   // UNICODE_TO_GBK[42326] := 16#9DDE;
   // UNICODE_TO_GBK[42327] := 16#FA7B;
   // UNICODE_TO_GBK[42328] := 16#9DDF;
   // UNICODE_TO_GBK[42329] := 16#FA7C;
   // UNICODE_TO_GBK[42330] := 16#9DE0;
   // UNICODE_TO_GBK[42331] := 16#FA7D;
   // UNICODE_TO_GBK[42332] := 16#9DE1;
   // UNICODE_TO_GBK[42333] := 16#FA7E;
   // UNICODE_TO_GBK[42334] := 16#9DE2;
   // UNICODE_TO_GBK[42335] := 16#FA80;
   // UNICODE_TO_GBK[42336] := 16#9DE3;
   // UNICODE_TO_GBK[42337] := 16#FA81;
   // UNICODE_TO_GBK[42338] := 16#9DE4;
   // UNICODE_TO_GBK[42339] := 16#FA82;
   // UNICODE_TO_GBK[42340] := 16#9DE5;
   // UNICODE_TO_GBK[42341] := 16#FA83;
   // UNICODE_TO_GBK[42342] := 16#9DE6;
   // UNICODE_TO_GBK[42343] := 16#FA84;
   // UNICODE_TO_GBK[42344] := 16#9DE7;
   // UNICODE_TO_GBK[42345] := 16#FA85;
   // UNICODE_TO_GBK[42346] := 16#9DE8;
   // UNICODE_TO_GBK[42347] := 16#FA86;
   // UNICODE_TO_GBK[42348] := 16#9DE9;
   // UNICODE_TO_GBK[42349] := 16#FA87;
   // UNICODE_TO_GBK[42350] := 16#9DEA;
   // UNICODE_TO_GBK[42351] := 16#FA88;
   // UNICODE_TO_GBK[42352] := 16#9DEB;
   // UNICODE_TO_GBK[42353] := 16#FA89;
   // UNICODE_TO_GBK[42354] := 16#9DEC;
   // UNICODE_TO_GBK[42355] := 16#FA8A;
   // UNICODE_TO_GBK[42356] := 16#9DED;
   // UNICODE_TO_GBK[42357] := 16#FA8B;
   // UNICODE_TO_GBK[42358] := 16#9DEE;
   // UNICODE_TO_GBK[42359] := 16#FA8C;
   // UNICODE_TO_GBK[42360] := 16#9DEF;
   // UNICODE_TO_GBK[42361] := 16#FA8D;
   // UNICODE_TO_GBK[42362] := 16#9DF0;
   // UNICODE_TO_GBK[42363] := 16#FA8E;
   // UNICODE_TO_GBK[42364] := 16#9DF1;
   // UNICODE_TO_GBK[42365] := 16#FA8F;
   // UNICODE_TO_GBK[42366] := 16#9DF2;
   // UNICODE_TO_GBK[42367] := 16#FA90;
   // UNICODE_TO_GBK[42368] := 16#9DF3;
   // UNICODE_TO_GBK[42369] := 16#FA91;
   // UNICODE_TO_GBK[42370] := 16#9DF4;
   // UNICODE_TO_GBK[42371] := 16#FA92;
   // UNICODE_TO_GBK[42372] := 16#9DF5;
   // UNICODE_TO_GBK[42373] := 16#FA93;
   // UNICODE_TO_GBK[42374] := 16#9DF6;
   // UNICODE_TO_GBK[42375] := 16#FA94;
   // UNICODE_TO_GBK[42376] := 16#9DF7;
   // UNICODE_TO_GBK[42377] := 16#FA95;
   // UNICODE_TO_GBK[42378] := 16#9DF8;
   // UNICODE_TO_GBK[42379] := 16#FA96;
   // UNICODE_TO_GBK[42380] := 16#9DF9;
   // UNICODE_TO_GBK[42381] := 16#FA97;
   // UNICODE_TO_GBK[42382] := 16#9DFA;
   // UNICODE_TO_GBK[42383] := 16#FA98;
   // UNICODE_TO_GBK[42384] := 16#9DFB;
   // UNICODE_TO_GBK[42385] := 16#FA99;
   // UNICODE_TO_GBK[42386] := 16#9DFC;
   // UNICODE_TO_GBK[42387] := 16#FA9A;
   // UNICODE_TO_GBK[42388] := 16#9DFD;
   // UNICODE_TO_GBK[42389] := 16#FA9B;
   // UNICODE_TO_GBK[42390] := 16#9DFE;
   // UNICODE_TO_GBK[42391] := 16#FA9C;
   // UNICODE_TO_GBK[42392] := 16#9DFF;
   // UNICODE_TO_GBK[42393] := 16#FA9D;
   // UNICODE_TO_GBK[42394] := 16#9E00;
   // UNICODE_TO_GBK[42395] := 16#FA9E;
   // UNICODE_TO_GBK[42396] := 16#9E01;
   // UNICODE_TO_GBK[42397] := 16#FA9F;
   // UNICODE_TO_GBK[42398] := 16#9E02;
   // UNICODE_TO_GBK[42399] := 16#FAA0;
   // UNICODE_TO_GBK[42400] := 16#9E03;
   // UNICODE_TO_GBK[42401] := 16#FB40;
   // UNICODE_TO_GBK[42402] := 16#9E04;
   // UNICODE_TO_GBK[42403] := 16#FB41;
   // UNICODE_TO_GBK[42404] := 16#9E05;
   // UNICODE_TO_GBK[42405] := 16#FB42;
   // UNICODE_TO_GBK[42406] := 16#9E06;
   // UNICODE_TO_GBK[42407] := 16#FB43;
   // UNICODE_TO_GBK[42408] := 16#9E07;
   // UNICODE_TO_GBK[42409] := 16#FB44;
   // UNICODE_TO_GBK[42410] := 16#9E08;
   // UNICODE_TO_GBK[42411] := 16#FB45;
   // UNICODE_TO_GBK[42412] := 16#9E09;
   // UNICODE_TO_GBK[42413] := 16#FB46;
   // UNICODE_TO_GBK[42414] := 16#9E0A;
   // UNICODE_TO_GBK[42415] := 16#FB47;
   // UNICODE_TO_GBK[42416] := 16#9E0B;
   // UNICODE_TO_GBK[42417] := 16#FB48;
   // UNICODE_TO_GBK[42418] := 16#9E0C;
   // UNICODE_TO_GBK[42419] := 16#FB49;
   // UNICODE_TO_GBK[42420] := 16#9E0D;
   // UNICODE_TO_GBK[42421] := 16#FB4A;
   // UNICODE_TO_GBK[42422] := 16#9E0E;
   // UNICODE_TO_GBK[42423] := 16#FB4B;
   // UNICODE_TO_GBK[42424] := 16#9E0F;
   // UNICODE_TO_GBK[42425] := 16#FB4C;
   // UNICODE_TO_GBK[42426] := 16#9E10;
   // UNICODE_TO_GBK[42427] := 16#FB4D;
   // UNICODE_TO_GBK[42428] := 16#9E11;
   // UNICODE_TO_GBK[42429] := 16#FB4E;
   // UNICODE_TO_GBK[42430] := 16#9E12;
   // UNICODE_TO_GBK[42431] := 16#FB4F;
   // UNICODE_TO_GBK[42432] := 16#9E13;
   // UNICODE_TO_GBK[42433] := 16#FB50;
   // UNICODE_TO_GBK[42434] := 16#9E14;
   // UNICODE_TO_GBK[42435] := 16#FB51;
   // UNICODE_TO_GBK[42436] := 16#9E15;
   // UNICODE_TO_GBK[42437] := 16#FB52;
   // UNICODE_TO_GBK[42438] := 16#9E16;
   // UNICODE_TO_GBK[42439] := 16#FB53;
   // UNICODE_TO_GBK[42440] := 16#9E17;
   // UNICODE_TO_GBK[42441] := 16#FB54;
   // UNICODE_TO_GBK[42442] := 16#9E18;
   // UNICODE_TO_GBK[42443] := 16#FB55;
   // UNICODE_TO_GBK[42444] := 16#9E19;
   // UNICODE_TO_GBK[42445] := 16#FB56;
   // UNICODE_TO_GBK[42446] := 16#9E1A;
   // UNICODE_TO_GBK[42447] := 16#FB57;
   // UNICODE_TO_GBK[42448] := 16#9E1B;
   // UNICODE_TO_GBK[42449] := 16#FB58;
   // UNICODE_TO_GBK[42450] := 16#9E1C;
   // UNICODE_TO_GBK[42451] := 16#FB59;
   // UNICODE_TO_GBK[42452] := 16#9E1D;
   // UNICODE_TO_GBK[42453] := 16#FB5A;
   // UNICODE_TO_GBK[42454] := 16#9E1E;
   // UNICODE_TO_GBK[42455] := 16#FB5B;
   // UNICODE_TO_GBK[42456] := 16#9E1F;
   // UNICODE_TO_GBK[42457] := 16#C4F1;
   // UNICODE_TO_GBK[42458] := 16#9E20;
   // UNICODE_TO_GBK[42459] := 16#F0AF;
   // UNICODE_TO_GBK[42460] := 16#9E21;
   // UNICODE_TO_GBK[42461] := 16#BCA6;
   // UNICODE_TO_GBK[42462] := 16#9E22;
   // UNICODE_TO_GBK[42463] := 16#F0B0;
   // UNICODE_TO_GBK[42464] := 16#9E23;
   // UNICODE_TO_GBK[42465] := 16#C3F9;
   // UNICODE_TO_GBK[42466] := 16#9E24;
   // UNICODE_TO_GBK[42467] := 16#FB5C;
   // UNICODE_TO_GBK[42468] := 16#9E25;
   // UNICODE_TO_GBK[42469] := 16#C5B8;
   // UNICODE_TO_GBK[42470] := 16#9E26;
   // UNICODE_TO_GBK[42471] := 16#D1BB;
   // UNICODE_TO_GBK[42472] := 16#9E27;
   // UNICODE_TO_GBK[42473] := 16#FB5D;
   // UNICODE_TO_GBK[42474] := 16#9E28;
   // UNICODE_TO_GBK[42475] := 16#F0B1;
   // UNICODE_TO_GBK[42476] := 16#9E29;
   // UNICODE_TO_GBK[42477] := 16#F0B2;
   // UNICODE_TO_GBK[42478] := 16#9E2A;
   // UNICODE_TO_GBK[42479] := 16#F0B3;
   // UNICODE_TO_GBK[42480] := 16#9E2B;
   // UNICODE_TO_GBK[42481] := 16#F0B4;
   // UNICODE_TO_GBK[42482] := 16#9E2C;
   // UNICODE_TO_GBK[42483] := 16#F0B5;
   // UNICODE_TO_GBK[42484] := 16#9E2D;
   // UNICODE_TO_GBK[42485] := 16#D1BC;
   // UNICODE_TO_GBK[42486] := 16#9E2E;
   // UNICODE_TO_GBK[42487] := 16#FB5E;
   // UNICODE_TO_GBK[42488] := 16#9E2F;
   // UNICODE_TO_GBK[42489] := 16#D1EC;
   // UNICODE_TO_GBK[42490] := 16#9E30;
   // UNICODE_TO_GBK[42491] := 16#FB5F;
   // UNICODE_TO_GBK[42492] := 16#9E31;
   // UNICODE_TO_GBK[42493] := 16#F0B7;
   // UNICODE_TO_GBK[42494] := 16#9E32;
   // UNICODE_TO_GBK[42495] := 16#F0B6;
   // UNICODE_TO_GBK[42496] := 16#9E33;
   // UNICODE_TO_GBK[42497] := 16#D4A7;
   // UNICODE_TO_GBK[42498] := 16#9E34;
   // UNICODE_TO_GBK[42499] := 16#FB60;
   // UNICODE_TO_GBK[42500] := 16#9E35;
   // UNICODE_TO_GBK[42501] := 16#CDD2;
   // UNICODE_TO_GBK[42502] := 16#9E36;
   // UNICODE_TO_GBK[42503] := 16#F0B8;
   // UNICODE_TO_GBK[42504] := 16#9E37;
   // UNICODE_TO_GBK[42505] := 16#F0BA;
   // UNICODE_TO_GBK[42506] := 16#9E38;
   // UNICODE_TO_GBK[42507] := 16#F0B9;
   // UNICODE_TO_GBK[42508] := 16#9E39;
   // UNICODE_TO_GBK[42509] := 16#F0BB;
   // UNICODE_TO_GBK[42510] := 16#9E3A;
   // UNICODE_TO_GBK[42511] := 16#F0BC;
   // UNICODE_TO_GBK[42512] := 16#9E3B;
   // UNICODE_TO_GBK[42513] := 16#FB61;
   // UNICODE_TO_GBK[42514] := 16#9E3C;
   // UNICODE_TO_GBK[42515] := 16#FB62;
   // UNICODE_TO_GBK[42516] := 16#9E3D;
   // UNICODE_TO_GBK[42517] := 16#B8EB;
   // UNICODE_TO_GBK[42518] := 16#9E3E;
   // UNICODE_TO_GBK[42519] := 16#F0BD;
   // UNICODE_TO_GBK[42520] := 16#9E3F;
   // UNICODE_TO_GBK[42521] := 16#BAE8;
   // UNICODE_TO_GBK[42522] := 16#9E40;
   // UNICODE_TO_GBK[42523] := 16#FB63;
   // UNICODE_TO_GBK[42524] := 16#9E41;
   // UNICODE_TO_GBK[42525] := 16#F0BE;
   // UNICODE_TO_GBK[42526] := 16#9E42;
   // UNICODE_TO_GBK[42527] := 16#F0BF;
   // UNICODE_TO_GBK[42528] := 16#9E43;
   // UNICODE_TO_GBK[42529] := 16#BEE9;
   // UNICODE_TO_GBK[42530] := 16#9E44;
   // UNICODE_TO_GBK[42531] := 16#F0C0;
   // UNICODE_TO_GBK[42532] := 16#9E45;
   // UNICODE_TO_GBK[42533] := 16#B6EC;
   // UNICODE_TO_GBK[42534] := 16#9E46;
   // UNICODE_TO_GBK[42535] := 16#F0C1;
   // UNICODE_TO_GBK[42536] := 16#9E47;
   // UNICODE_TO_GBK[42537] := 16#F0C2;
   // UNICODE_TO_GBK[42538] := 16#9E48;
   // UNICODE_TO_GBK[42539] := 16#F0C3;
   // UNICODE_TO_GBK[42540] := 16#9E49;
   // UNICODE_TO_GBK[42541] := 16#F0C4;
   // UNICODE_TO_GBK[42542] := 16#9E4A;
   // UNICODE_TO_GBK[42543] := 16#C8B5;
   // UNICODE_TO_GBK[42544] := 16#9E4B;
   // UNICODE_TO_GBK[42545] := 16#F0C5;
   // UNICODE_TO_GBK[42546] := 16#9E4C;
   // UNICODE_TO_GBK[42547] := 16#F0C6;
   // UNICODE_TO_GBK[42548] := 16#9E4D;
   // UNICODE_TO_GBK[42549] := 16#FB64;
   // UNICODE_TO_GBK[42550] := 16#9E4E;
   // UNICODE_TO_GBK[42551] := 16#F0C7;
   // UNICODE_TO_GBK[42552] := 16#9E4F;
   // UNICODE_TO_GBK[42553] := 16#C5F4;
   // UNICODE_TO_GBK[42554] := 16#9E50;
   // UNICODE_TO_GBK[42555] := 16#FB65;
   // UNICODE_TO_GBK[42556] := 16#9E51;
   // UNICODE_TO_GBK[42557] := 16#F0C8;
   // UNICODE_TO_GBK[42558] := 16#9E52;
   // UNICODE_TO_GBK[42559] := 16#FB66;
   // UNICODE_TO_GBK[42560] := 16#9E53;
   // UNICODE_TO_GBK[42561] := 16#FB67;
   // UNICODE_TO_GBK[42562] := 16#9E54;
   // UNICODE_TO_GBK[42563] := 16#FB68;
   // UNICODE_TO_GBK[42564] := 16#9E55;
   // UNICODE_TO_GBK[42565] := 16#F0C9;
   // UNICODE_TO_GBK[42566] := 16#9E56;
   // UNICODE_TO_GBK[42567] := 16#FB69;
   // UNICODE_TO_GBK[42568] := 16#9E57;
   // UNICODE_TO_GBK[42569] := 16#F0CA;
   // UNICODE_TO_GBK[42570] := 16#9E58;
   // UNICODE_TO_GBK[42571] := 16#F7BD;
   // UNICODE_TO_GBK[42572] := 16#9E59;
   // UNICODE_TO_GBK[42573] := 16#FB6A;
   // UNICODE_TO_GBK[42574] := 16#9E5A;
   // UNICODE_TO_GBK[42575] := 16#F0CB;
   // UNICODE_TO_GBK[42576] := 16#9E5B;
   // UNICODE_TO_GBK[42577] := 16#F0CC;
   // UNICODE_TO_GBK[42578] := 16#9E5C;
   // UNICODE_TO_GBK[42579] := 16#F0CD;
   // UNICODE_TO_GBK[42580] := 16#9E5D;
   // UNICODE_TO_GBK[42581] := 16#FB6B;
   // UNICODE_TO_GBK[42582] := 16#9E5E;
   // UNICODE_TO_GBK[42583] := 16#F0CE;
   // UNICODE_TO_GBK[42584] := 16#9E5F;
   // UNICODE_TO_GBK[42585] := 16#FB6C;
   // UNICODE_TO_GBK[42586] := 16#9E60;
   // UNICODE_TO_GBK[42587] := 16#FB6D;
   // UNICODE_TO_GBK[42588] := 16#9E61;
   // UNICODE_TO_GBK[42589] := 16#FB6E;
   // UNICODE_TO_GBK[42590] := 16#9E62;
   // UNICODE_TO_GBK[42591] := 16#FB6F;
   // UNICODE_TO_GBK[42592] := 16#9E63;
   // UNICODE_TO_GBK[42593] := 16#F0CF;
   // UNICODE_TO_GBK[42594] := 16#9E64;
   // UNICODE_TO_GBK[42595] := 16#BAD7;
   // UNICODE_TO_GBK[42596] := 16#9E65;
   // UNICODE_TO_GBK[42597] := 16#FB70;
   // UNICODE_TO_GBK[42598] := 16#9E66;
   // UNICODE_TO_GBK[42599] := 16#F0D0;
   // UNICODE_TO_GBK[42600] := 16#9E67;
   // UNICODE_TO_GBK[42601] := 16#F0D1;
   // UNICODE_TO_GBK[42602] := 16#9E68;
   // UNICODE_TO_GBK[42603] := 16#F0D2;
   // UNICODE_TO_GBK[42604] := 16#9E69;
   // UNICODE_TO_GBK[42605] := 16#F0D3;
   // UNICODE_TO_GBK[42606] := 16#9E6A;
   // UNICODE_TO_GBK[42607] := 16#F0D4;
   // UNICODE_TO_GBK[42608] := 16#9E6B;
   // UNICODE_TO_GBK[42609] := 16#F0D5;
   // UNICODE_TO_GBK[42610] := 16#9E6C;
   // UNICODE_TO_GBK[42611] := 16#F0D6;
   // UNICODE_TO_GBK[42612] := 16#9E6D;
   // UNICODE_TO_GBK[42613] := 16#F0D8;
   // UNICODE_TO_GBK[42614] := 16#9E6E;
   // UNICODE_TO_GBK[42615] := 16#FB71;
   // UNICODE_TO_GBK[42616] := 16#9E6F;
   // UNICODE_TO_GBK[42617] := 16#FB72;
   // UNICODE_TO_GBK[42618] := 16#9E70;
   // UNICODE_TO_GBK[42619] := 16#D3A5;
   // UNICODE_TO_GBK[42620] := 16#9E71;
   // UNICODE_TO_GBK[42621] := 16#F0D7;
   // UNICODE_TO_GBK[42622] := 16#9E72;
   // UNICODE_TO_GBK[42623] := 16#FB73;
   // UNICODE_TO_GBK[42624] := 16#9E73;
   // UNICODE_TO_GBK[42625] := 16#F0D9;
   // UNICODE_TO_GBK[42626] := 16#9E74;
   // UNICODE_TO_GBK[42627] := 16#FB74;
   // UNICODE_TO_GBK[42628] := 16#9E75;
   // UNICODE_TO_GBK[42629] := 16#FB75;
   // UNICODE_TO_GBK[42630] := 16#9E76;
   // UNICODE_TO_GBK[42631] := 16#FB76;
   // UNICODE_TO_GBK[42632] := 16#9E77;
   // UNICODE_TO_GBK[42633] := 16#FB77;
   // UNICODE_TO_GBK[42634] := 16#9E78;
   // UNICODE_TO_GBK[42635] := 16#FB78;
   // UNICODE_TO_GBK[42636] := 16#9E79;
   // UNICODE_TO_GBK[42637] := 16#FB79;
   // UNICODE_TO_GBK[42638] := 16#9E7A;
   // UNICODE_TO_GBK[42639] := 16#FB7A;
   // UNICODE_TO_GBK[42640] := 16#9E7B;
   // UNICODE_TO_GBK[42641] := 16#FB7B;
   // UNICODE_TO_GBK[42642] := 16#9E7C;
   // UNICODE_TO_GBK[42643] := 16#FB7C;
   // UNICODE_TO_GBK[42644] := 16#9E7D;
   // UNICODE_TO_GBK[42645] := 16#FB7D;
   // UNICODE_TO_GBK[42646] := 16#9E7E;
   // UNICODE_TO_GBK[42647] := 16#F5BA;
   // UNICODE_TO_GBK[42648] := 16#9E7F;
   // UNICODE_TO_GBK[42649] := 16#C2B9;
   // UNICODE_TO_GBK[42650] := 16#9E80;
   // UNICODE_TO_GBK[42651] := 16#FB7E;
   // UNICODE_TO_GBK[42652] := 16#9E81;
   // UNICODE_TO_GBK[42653] := 16#FB80;
   // UNICODE_TO_GBK[42654] := 16#9E82;
   // UNICODE_TO_GBK[42655] := 16#F7E4;
   // UNICODE_TO_GBK[42656] := 16#9E83;
   // UNICODE_TO_GBK[42657] := 16#FB81;
   // UNICODE_TO_GBK[42658] := 16#9E84;
   // UNICODE_TO_GBK[42659] := 16#FB82;
   // UNICODE_TO_GBK[42660] := 16#9E85;
   // UNICODE_TO_GBK[42661] := 16#FB83;
   // UNICODE_TO_GBK[42662] := 16#9E86;
   // UNICODE_TO_GBK[42663] := 16#FB84;
   // UNICODE_TO_GBK[42664] := 16#9E87;
   // UNICODE_TO_GBK[42665] := 16#F7E5;
   // UNICODE_TO_GBK[42666] := 16#9E88;
   // UNICODE_TO_GBK[42667] := 16#F7E6;
   // UNICODE_TO_GBK[42668] := 16#9E89;
   // UNICODE_TO_GBK[42669] := 16#FB85;
   // UNICODE_TO_GBK[42670] := 16#9E8A;
   // UNICODE_TO_GBK[42671] := 16#FB86;
   // UNICODE_TO_GBK[42672] := 16#9E8B;
   // UNICODE_TO_GBK[42673] := 16#F7E7;
   // UNICODE_TO_GBK[42674] := 16#9E8C;
   // UNICODE_TO_GBK[42675] := 16#FB87;
   // UNICODE_TO_GBK[42676] := 16#9E8D;
   // UNICODE_TO_GBK[42677] := 16#FB88;
   // UNICODE_TO_GBK[42678] := 16#9E8E;
   // UNICODE_TO_GBK[42679] := 16#FB89;
   // UNICODE_TO_GBK[42680] := 16#9E8F;
   // UNICODE_TO_GBK[42681] := 16#FB8A;
   // UNICODE_TO_GBK[42682] := 16#9E90;
   // UNICODE_TO_GBK[42683] := 16#FB8B;
   // UNICODE_TO_GBK[42684] := 16#9E91;
   // UNICODE_TO_GBK[42685] := 16#FB8C;
   // UNICODE_TO_GBK[42686] := 16#9E92;
   // UNICODE_TO_GBK[42687] := 16#F7E8;
   // UNICODE_TO_GBK[42688] := 16#9E93;
   // UNICODE_TO_GBK[42689] := 16#C2B4;
   // UNICODE_TO_GBK[42690] := 16#9E94;
   // UNICODE_TO_GBK[42691] := 16#FB8D;
   // UNICODE_TO_GBK[42692] := 16#9E95;
   // UNICODE_TO_GBK[42693] := 16#FB8E;
   // UNICODE_TO_GBK[42694] := 16#9E96;
   // UNICODE_TO_GBK[42695] := 16#FB8F;
   // UNICODE_TO_GBK[42696] := 16#9E97;
   // UNICODE_TO_GBK[42697] := 16#FB90;
   // UNICODE_TO_GBK[42698] := 16#9E98;
   // UNICODE_TO_GBK[42699] := 16#FB91;
   // UNICODE_TO_GBK[42700] := 16#9E99;
   // UNICODE_TO_GBK[42701] := 16#FB92;
   // UNICODE_TO_GBK[42702] := 16#9E9A;
   // UNICODE_TO_GBK[42703] := 16#FB93;
   // UNICODE_TO_GBK[42704] := 16#9E9B;
   // UNICODE_TO_GBK[42705] := 16#FB94;
   // UNICODE_TO_GBK[42706] := 16#9E9C;
   // UNICODE_TO_GBK[42707] := 16#FB95;
   // UNICODE_TO_GBK[42708] := 16#9E9D;
   // UNICODE_TO_GBK[42709] := 16#F7EA;
   // UNICODE_TO_GBK[42710] := 16#9E9E;
   // UNICODE_TO_GBK[42711] := 16#FB96;
   // UNICODE_TO_GBK[42712] := 16#9E9F;
   // UNICODE_TO_GBK[42713] := 16#F7EB;
   // UNICODE_TO_GBK[42714] := 16#9EA0;
   // UNICODE_TO_GBK[42715] := 16#FB97;
   // UNICODE_TO_GBK[42716] := 16#9EA1;
   // UNICODE_TO_GBK[42717] := 16#FB98;
   // UNICODE_TO_GBK[42718] := 16#9EA2;
   // UNICODE_TO_GBK[42719] := 16#FB99;
   // UNICODE_TO_GBK[42720] := 16#9EA3;
   // UNICODE_TO_GBK[42721] := 16#FB9A;
   // UNICODE_TO_GBK[42722] := 16#9EA4;
   // UNICODE_TO_GBK[42723] := 16#FB9B;
   // UNICODE_TO_GBK[42724] := 16#9EA5;
   // UNICODE_TO_GBK[42725] := 16#FB9C;
   // UNICODE_TO_GBK[42726] := 16#9EA6;
   // UNICODE_TO_GBK[42727] := 16#C2F3;
   // UNICODE_TO_GBK[42728] := 16#9EA7;
   // UNICODE_TO_GBK[42729] := 16#FB9D;
   // UNICODE_TO_GBK[42730] := 16#9EA8;
   // UNICODE_TO_GBK[42731] := 16#FB9E;
   // UNICODE_TO_GBK[42732] := 16#9EA9;
   // UNICODE_TO_GBK[42733] := 16#FB9F;
   // UNICODE_TO_GBK[42734] := 16#9EAA;
   // UNICODE_TO_GBK[42735] := 16#FBA0;
   // UNICODE_TO_GBK[42736] := 16#9EAB;
   // UNICODE_TO_GBK[42737] := 16#FC40;
   // UNICODE_TO_GBK[42738] := 16#9EAC;
   // UNICODE_TO_GBK[42739] := 16#FC41;
   // UNICODE_TO_GBK[42740] := 16#9EAD;
   // UNICODE_TO_GBK[42741] := 16#FC42;
   // UNICODE_TO_GBK[42742] := 16#9EAE;
   // UNICODE_TO_GBK[42743] := 16#FC43;
   // UNICODE_TO_GBK[42744] := 16#9EAF;
   // UNICODE_TO_GBK[42745] := 16#FC44;
   // UNICODE_TO_GBK[42746] := 16#9EB0;
   // UNICODE_TO_GBK[42747] := 16#FC45;
   // UNICODE_TO_GBK[42748] := 16#9EB1;
   // UNICODE_TO_GBK[42749] := 16#FC46;
   // UNICODE_TO_GBK[42750] := 16#9EB2;
   // UNICODE_TO_GBK[42751] := 16#FC47;
   // UNICODE_TO_GBK[42752] := 16#9EB3;
   // UNICODE_TO_GBK[42753] := 16#FC48;
   // UNICODE_TO_GBK[42754] := 16#9EB4;
   // UNICODE_TO_GBK[42755] := 16#F4F0;
   // UNICODE_TO_GBK[42756] := 16#9EB5;
   // UNICODE_TO_GBK[42757] := 16#FC49;
   // UNICODE_TO_GBK[42758] := 16#9EB6;
   // UNICODE_TO_GBK[42759] := 16#FC4A;
   // UNICODE_TO_GBK[42760] := 16#9EB7;
   // UNICODE_TO_GBK[42761] := 16#FC4B;
   // UNICODE_TO_GBK[42762] := 16#9EB8;
   // UNICODE_TO_GBK[42763] := 16#F4EF;
   // UNICODE_TO_GBK[42764] := 16#9EB9;
   // UNICODE_TO_GBK[42765] := 16#FC4C;
   // UNICODE_TO_GBK[42766] := 16#9EBA;
   // UNICODE_TO_GBK[42767] := 16#FC4D;
   // UNICODE_TO_GBK[42768] := 16#9EBB;
   // UNICODE_TO_GBK[42769] := 16#C2E9;
   // UNICODE_TO_GBK[42770] := 16#9EBC;
   // UNICODE_TO_GBK[42771] := 16#FC4E;
   // UNICODE_TO_GBK[42772] := 16#9EBD;
   // UNICODE_TO_GBK[42773] := 16#F7E1;
   // UNICODE_TO_GBK[42774] := 16#9EBE;
   // UNICODE_TO_GBK[42775] := 16#F7E2;
   // UNICODE_TO_GBK[42776] := 16#9EBF;
   // UNICODE_TO_GBK[42777] := 16#FC4F;
   // UNICODE_TO_GBK[42778] := 16#9EC0;
   // UNICODE_TO_GBK[42779] := 16#FC50;
   // UNICODE_TO_GBK[42780] := 16#9EC1;
   // UNICODE_TO_GBK[42781] := 16#FC51;
   // UNICODE_TO_GBK[42782] := 16#9EC2;
   // UNICODE_TO_GBK[42783] := 16#FC52;
   // UNICODE_TO_GBK[42784] := 16#9EC3;
   // UNICODE_TO_GBK[42785] := 16#FC53;
   // UNICODE_TO_GBK[42786] := 16#9EC4;
   // UNICODE_TO_GBK[42787] := 16#BBC6;
   // UNICODE_TO_GBK[42788] := 16#9EC5;
   // UNICODE_TO_GBK[42789] := 16#FC54;
   // UNICODE_TO_GBK[42790] := 16#9EC6;
   // UNICODE_TO_GBK[42791] := 16#FC55;
   // UNICODE_TO_GBK[42792] := 16#9EC7;
   // UNICODE_TO_GBK[42793] := 16#FC56;
   // UNICODE_TO_GBK[42794] := 16#9EC8;
   // UNICODE_TO_GBK[42795] := 16#FC57;
   // UNICODE_TO_GBK[42796] := 16#9EC9;
   // UNICODE_TO_GBK[42797] := 16#D9E4;
   // UNICODE_TO_GBK[42798] := 16#9ECA;
   // UNICODE_TO_GBK[42799] := 16#FC58;
   // UNICODE_TO_GBK[42800] := 16#9ECB;
   // UNICODE_TO_GBK[42801] := 16#FC59;
   // UNICODE_TO_GBK[42802] := 16#9ECC;
   // UNICODE_TO_GBK[42803] := 16#FC5A;
   // UNICODE_TO_GBK[42804] := 16#9ECD;
   // UNICODE_TO_GBK[42805] := 16#CAF2;
   // UNICODE_TO_GBK[42806] := 16#9ECE;
   // UNICODE_TO_GBK[42807] := 16#C0E8;
   // UNICODE_TO_GBK[42808] := 16#9ECF;
   // UNICODE_TO_GBK[42809] := 16#F0A4;
   // UNICODE_TO_GBK[42810] := 16#9ED0;
   // UNICODE_TO_GBK[42811] := 16#FC5B;
   // UNICODE_TO_GBK[42812] := 16#9ED1;
   // UNICODE_TO_GBK[42813] := 16#BADA;
   // UNICODE_TO_GBK[42814] := 16#9ED2;
   // UNICODE_TO_GBK[42815] := 16#FC5C;
   // UNICODE_TO_GBK[42816] := 16#9ED3;
   // UNICODE_TO_GBK[42817] := 16#FC5D;
   // UNICODE_TO_GBK[42818] := 16#9ED4;
   // UNICODE_TO_GBK[42819] := 16#C7AD;
   // UNICODE_TO_GBK[42820] := 16#9ED5;
   // UNICODE_TO_GBK[42821] := 16#FC5E;
   // UNICODE_TO_GBK[42822] := 16#9ED6;
   // UNICODE_TO_GBK[42823] := 16#FC5F;
   // UNICODE_TO_GBK[42824] := 16#9ED7;
   // UNICODE_TO_GBK[42825] := 16#FC60;
   // UNICODE_TO_GBK[42826] := 16#9ED8;
   // UNICODE_TO_GBK[42827] := 16#C4AC;
   // UNICODE_TO_GBK[42828] := 16#9ED9;
   // UNICODE_TO_GBK[42829] := 16#FC61;
   // UNICODE_TO_GBK[42830] := 16#9EDA;
   // UNICODE_TO_GBK[42831] := 16#FC62;
   // UNICODE_TO_GBK[42832] := 16#9EDB;
   // UNICODE_TO_GBK[42833] := 16#F7EC;
   // UNICODE_TO_GBK[42834] := 16#9EDC;
   // UNICODE_TO_GBK[42835] := 16#F7ED;
   // UNICODE_TO_GBK[42836] := 16#9EDD;
   // UNICODE_TO_GBK[42837] := 16#F7EE;
   // UNICODE_TO_GBK[42838] := 16#9EDE;
   // UNICODE_TO_GBK[42839] := 16#FC63;
   // UNICODE_TO_GBK[42840] := 16#9EDF;
   // UNICODE_TO_GBK[42841] := 16#F7F0;
   // UNICODE_TO_GBK[42842] := 16#9EE0;
   // UNICODE_TO_GBK[42843] := 16#F7EF;
   // UNICODE_TO_GBK[42844] := 16#9EE1;
   // UNICODE_TO_GBK[42845] := 16#FC64;
   // UNICODE_TO_GBK[42846] := 16#9EE2;
   // UNICODE_TO_GBK[42847] := 16#F7F1;
   // UNICODE_TO_GBK[42848] := 16#9EE3;
   // UNICODE_TO_GBK[42849] := 16#FC65;
   // UNICODE_TO_GBK[42850] := 16#9EE4;
   // UNICODE_TO_GBK[42851] := 16#FC66;
   // UNICODE_TO_GBK[42852] := 16#9EE5;
   // UNICODE_TO_GBK[42853] := 16#F7F4;
   // UNICODE_TO_GBK[42854] := 16#9EE6;
   // UNICODE_TO_GBK[42855] := 16#FC67;
   // UNICODE_TO_GBK[42856] := 16#9EE7;
   // UNICODE_TO_GBK[42857] := 16#F7F3;
   // UNICODE_TO_GBK[42858] := 16#9EE8;
   // UNICODE_TO_GBK[42859] := 16#FC68;
   // UNICODE_TO_GBK[42860] := 16#9EE9;
   // UNICODE_TO_GBK[42861] := 16#F7F2;
   // UNICODE_TO_GBK[42862] := 16#9EEA;
   // UNICODE_TO_GBK[42863] := 16#F7F5;
   // UNICODE_TO_GBK[42864] := 16#9EEB;
   // UNICODE_TO_GBK[42865] := 16#FC69;
   // UNICODE_TO_GBK[42866] := 16#9EEC;
   // UNICODE_TO_GBK[42867] := 16#FC6A;
   // UNICODE_TO_GBK[42868] := 16#9EED;
   // UNICODE_TO_GBK[42869] := 16#FC6B;
   // UNICODE_TO_GBK[42870] := 16#9EEE;
   // UNICODE_TO_GBK[42871] := 16#FC6C;
   // UNICODE_TO_GBK[42872] := 16#9EEF;
   // UNICODE_TO_GBK[42873] := 16#F7F6;
   // UNICODE_TO_GBK[42874] := 16#9EF0;
   // UNICODE_TO_GBK[42875] := 16#FC6D;
   // UNICODE_TO_GBK[42876] := 16#9EF1;
   // UNICODE_TO_GBK[42877] := 16#FC6E;
   // UNICODE_TO_GBK[42878] := 16#9EF2;
   // UNICODE_TO_GBK[42879] := 16#FC6F;
   // UNICODE_TO_GBK[42880] := 16#9EF3;
   // UNICODE_TO_GBK[42881] := 16#FC70;
   // UNICODE_TO_GBK[42882] := 16#9EF4;
   // UNICODE_TO_GBK[42883] := 16#FC71;
   // UNICODE_TO_GBK[42884] := 16#9EF5;
   // UNICODE_TO_GBK[42885] := 16#FC72;
   // UNICODE_TO_GBK[42886] := 16#9EF6;
   // UNICODE_TO_GBK[42887] := 16#FC73;
   // UNICODE_TO_GBK[42888] := 16#9EF7;
   // UNICODE_TO_GBK[42889] := 16#FC74;
   // UNICODE_TO_GBK[42890] := 16#9EF8;
   // UNICODE_TO_GBK[42891] := 16#FC75;
   // UNICODE_TO_GBK[42892] := 16#9EF9;
   // UNICODE_TO_GBK[42893] := 16#EDE9;
   // UNICODE_TO_GBK[42894] := 16#9EFA;
   // UNICODE_TO_GBK[42895] := 16#FC76;
   // UNICODE_TO_GBK[42896] := 16#9EFB;
   // UNICODE_TO_GBK[42897] := 16#EDEA;
   // UNICODE_TO_GBK[42898] := 16#9EFC;
   // UNICODE_TO_GBK[42899] := 16#EDEB;
   // UNICODE_TO_GBK[42900] := 16#9EFD;
   // UNICODE_TO_GBK[42901] := 16#FC77;
   // UNICODE_TO_GBK[42902] := 16#9EFE;
   // UNICODE_TO_GBK[42903] := 16#F6BC;
   // UNICODE_TO_GBK[42904] := 16#9EFF;
   // UNICODE_TO_GBK[42905] := 16#FC78;
   // UNICODE_TO_GBK[42906] := 16#9F00;
   // UNICODE_TO_GBK[42907] := 16#FC79;
   // UNICODE_TO_GBK[42908] := 16#9F01;
   // UNICODE_TO_GBK[42909] := 16#FC7A;
   // UNICODE_TO_GBK[42910] := 16#9F02;
   // UNICODE_TO_GBK[42911] := 16#FC7B;
   // UNICODE_TO_GBK[42912] := 16#9F03;
   // UNICODE_TO_GBK[42913] := 16#FC7C;
   // UNICODE_TO_GBK[42914] := 16#9F04;
   // UNICODE_TO_GBK[42915] := 16#FC7D;
   // UNICODE_TO_GBK[42916] := 16#9F05;
   // UNICODE_TO_GBK[42917] := 16#FC7E;
   // UNICODE_TO_GBK[42918] := 16#9F06;
   // UNICODE_TO_GBK[42919] := 16#FC80;
   // UNICODE_TO_GBK[42920] := 16#9F07;
   // UNICODE_TO_GBK[42921] := 16#FC81;
   // UNICODE_TO_GBK[42922] := 16#9F08;
   // UNICODE_TO_GBK[42923] := 16#FC82;
   // UNICODE_TO_GBK[42924] := 16#9F09;
   // UNICODE_TO_GBK[42925] := 16#FC83;
   // UNICODE_TO_GBK[42926] := 16#9F0A;
   // UNICODE_TO_GBK[42927] := 16#FC84;
   // UNICODE_TO_GBK[42928] := 16#9F0B;
   // UNICODE_TO_GBK[42929] := 16#F6BD;
   // UNICODE_TO_GBK[42930] := 16#9F0C;
   // UNICODE_TO_GBK[42931] := 16#FC85;
   // UNICODE_TO_GBK[42932] := 16#9F0D;
   // UNICODE_TO_GBK[42933] := 16#F6BE;
   // UNICODE_TO_GBK[42934] := 16#9F0E;
   // UNICODE_TO_GBK[42935] := 16#B6A6;
   // UNICODE_TO_GBK[42936] := 16#9F0F;
   // UNICODE_TO_GBK[42937] := 16#FC86;
   // UNICODE_TO_GBK[42938] := 16#9F10;
   // UNICODE_TO_GBK[42939] := 16#D8BE;
   // UNICODE_TO_GBK[42940] := 16#9F11;
   // UNICODE_TO_GBK[42941] := 16#FC87;
   // UNICODE_TO_GBK[42942] := 16#9F12;
   // UNICODE_TO_GBK[42943] := 16#FC88;
   // UNICODE_TO_GBK[42944] := 16#9F13;
   // UNICODE_TO_GBK[42945] := 16#B9C4;
   // UNICODE_TO_GBK[42946] := 16#9F14;
   // UNICODE_TO_GBK[42947] := 16#FC89;
   // UNICODE_TO_GBK[42948] := 16#9F15;
   // UNICODE_TO_GBK[42949] := 16#FC8A;
   // UNICODE_TO_GBK[42950] := 16#9F16;
   // UNICODE_TO_GBK[42951] := 16#FC8B;
   // UNICODE_TO_GBK[42952] := 16#9F17;
   // UNICODE_TO_GBK[42953] := 16#D8BB;
   // UNICODE_TO_GBK[42954] := 16#9F18;
   // UNICODE_TO_GBK[42955] := 16#FC8C;
   // UNICODE_TO_GBK[42956] := 16#9F19;
   // UNICODE_TO_GBK[42957] := 16#DCB1;
   // UNICODE_TO_GBK[42958] := 16#9F1A;
   // UNICODE_TO_GBK[42959] := 16#FC8D;
   // UNICODE_TO_GBK[42960] := 16#9F1B;
   // UNICODE_TO_GBK[42961] := 16#FC8E;
   // UNICODE_TO_GBK[42962] := 16#9F1C;
   // UNICODE_TO_GBK[42963] := 16#FC8F;
   // UNICODE_TO_GBK[42964] := 16#9F1D;
   // UNICODE_TO_GBK[42965] := 16#FC90;
   // UNICODE_TO_GBK[42966] := 16#9F1E;
   // UNICODE_TO_GBK[42967] := 16#FC91;
   // UNICODE_TO_GBK[42968] := 16#9F1F;
   // UNICODE_TO_GBK[42969] := 16#FC92;
   // UNICODE_TO_GBK[42970] := 16#9F20;
   // UNICODE_TO_GBK[42971] := 16#CAF3;
   // UNICODE_TO_GBK[42972] := 16#9F21;
   // UNICODE_TO_GBK[42973] := 16#FC93;
   // UNICODE_TO_GBK[42974] := 16#9F22;
   // UNICODE_TO_GBK[42975] := 16#F7F7;
   // UNICODE_TO_GBK[42976] := 16#9F23;
   // UNICODE_TO_GBK[42977] := 16#FC94;
   // UNICODE_TO_GBK[42978] := 16#9F24;
   // UNICODE_TO_GBK[42979] := 16#FC95;
   // UNICODE_TO_GBK[42980] := 16#9F25;
   // UNICODE_TO_GBK[42981] := 16#FC96;
   // UNICODE_TO_GBK[42982] := 16#9F26;
   // UNICODE_TO_GBK[42983] := 16#FC97;
   // UNICODE_TO_GBK[42984] := 16#9F27;
   // UNICODE_TO_GBK[42985] := 16#FC98;
   // UNICODE_TO_GBK[42986] := 16#9F28;
   // UNICODE_TO_GBK[42987] := 16#FC99;
   // UNICODE_TO_GBK[42988] := 16#9F29;
   // UNICODE_TO_GBK[42989] := 16#FC9A;
   // UNICODE_TO_GBK[42990] := 16#9F2A;
   // UNICODE_TO_GBK[42991] := 16#FC9B;
   // UNICODE_TO_GBK[42992] := 16#9F2B;
   // UNICODE_TO_GBK[42993] := 16#FC9C;
   // UNICODE_TO_GBK[42994] := 16#9F2C;
   // UNICODE_TO_GBK[42995] := 16#F7F8;
   // UNICODE_TO_GBK[42996] := 16#9F2D;
   // UNICODE_TO_GBK[42997] := 16#FC9D;
   // UNICODE_TO_GBK[42998] := 16#9F2E;
   // UNICODE_TO_GBK[42999] := 16#FC9E;
   // UNICODE_TO_GBK[43000] := 16#9F2F;
   // UNICODE_TO_GBK[43001] := 16#F7F9;
   // UNICODE_TO_GBK[43002] := 16#9F30;
   // UNICODE_TO_GBK[43003] := 16#FC9F;
   // UNICODE_TO_GBK[43004] := 16#9F31;
   // UNICODE_TO_GBK[43005] := 16#FCA0;
   // UNICODE_TO_GBK[43006] := 16#9F32;
   // UNICODE_TO_GBK[43007] := 16#FD40;
   // UNICODE_TO_GBK[43008] := 16#9F33;
   // UNICODE_TO_GBK[43009] := 16#FD41;
   // UNICODE_TO_GBK[43010] := 16#9F34;
   // UNICODE_TO_GBK[43011] := 16#FD42;
   // UNICODE_TO_GBK[43012] := 16#9F35;
   // UNICODE_TO_GBK[43013] := 16#FD43;
   // UNICODE_TO_GBK[43014] := 16#9F36;
   // UNICODE_TO_GBK[43015] := 16#FD44;
   // UNICODE_TO_GBK[43016] := 16#9F37;
   // UNICODE_TO_GBK[43017] := 16#F7FB;
   // UNICODE_TO_GBK[43018] := 16#9F38;
   // UNICODE_TO_GBK[43019] := 16#FD45;
   // UNICODE_TO_GBK[43020] := 16#9F39;
   // UNICODE_TO_GBK[43021] := 16#F7FA;
   // UNICODE_TO_GBK[43022] := 16#9F3A;
   // UNICODE_TO_GBK[43023] := 16#FD46;
   // UNICODE_TO_GBK[43024] := 16#9F3B;
   // UNICODE_TO_GBK[43025] := 16#B1C7;
   // UNICODE_TO_GBK[43026] := 16#9F3C;
   // UNICODE_TO_GBK[43027] := 16#FD47;
   // UNICODE_TO_GBK[43028] := 16#9F3D;
   // UNICODE_TO_GBK[43029] := 16#F7FC;
   // UNICODE_TO_GBK[43030] := 16#9F3E;
   // UNICODE_TO_GBK[43031] := 16#F7FD;
   // UNICODE_TO_GBK[43032] := 16#9F3F;
   // UNICODE_TO_GBK[43033] := 16#FD48;
   // UNICODE_TO_GBK[43034] := 16#9F40;
   // UNICODE_TO_GBK[43035] := 16#FD49;
   // UNICODE_TO_GBK[43036] := 16#9F41;
   // UNICODE_TO_GBK[43037] := 16#FD4A;
   // UNICODE_TO_GBK[43038] := 16#9F42;
   // UNICODE_TO_GBK[43039] := 16#FD4B;
   // UNICODE_TO_GBK[43040] := 16#9F43;
   // UNICODE_TO_GBK[43041] := 16#FD4C;
   // UNICODE_TO_GBK[43042] := 16#9F44;
   // UNICODE_TO_GBK[43043] := 16#F7FE;
   // UNICODE_TO_GBK[43044] := 16#9F45;
   // UNICODE_TO_GBK[43045] := 16#FD4D;
   // UNICODE_TO_GBK[43046] := 16#9F46;
   // UNICODE_TO_GBK[43047] := 16#FD4E;
   // UNICODE_TO_GBK[43048] := 16#9F47;
   // UNICODE_TO_GBK[43049] := 16#FD4F;
   // UNICODE_TO_GBK[43050] := 16#9F48;
   // UNICODE_TO_GBK[43051] := 16#FD50;
   // UNICODE_TO_GBK[43052] := 16#9F49;
   // UNICODE_TO_GBK[43053] := 16#FD51;
   // UNICODE_TO_GBK[43054] := 16#9F4A;
   // UNICODE_TO_GBK[43055] := 16#FD52;
   // UNICODE_TO_GBK[43056] := 16#9F4B;
   // UNICODE_TO_GBK[43057] := 16#FD53;
   // UNICODE_TO_GBK[43058] := 16#9F4C;
   // UNICODE_TO_GBK[43059] := 16#FD54;
   // UNICODE_TO_GBK[43060] := 16#9F4D;
   // UNICODE_TO_GBK[43061] := 16#FD55;
   // UNICODE_TO_GBK[43062] := 16#9F4E;
   // UNICODE_TO_GBK[43063] := 16#FD56;
   // UNICODE_TO_GBK[43064] := 16#9F4F;
   // UNICODE_TO_GBK[43065] := 16#FD57;
   // UNICODE_TO_GBK[43066] := 16#9F50;
   // UNICODE_TO_GBK[43067] := 16#C6EB;
   // UNICODE_TO_GBK[43068] := 16#9F51;
   // UNICODE_TO_GBK[43069] := 16#ECB4;
   // UNICODE_TO_GBK[43070] := 16#9F52;
   // UNICODE_TO_GBK[43071] := 16#FD58;
   // UNICODE_TO_GBK[43072] := 16#9F53;
   // UNICODE_TO_GBK[43073] := 16#FD59;
   // UNICODE_TO_GBK[43074] := 16#9F54;
   // UNICODE_TO_GBK[43075] := 16#FD5A;
   // UNICODE_TO_GBK[43076] := 16#9F55;
   // UNICODE_TO_GBK[43077] := 16#FD5B;
   // UNICODE_TO_GBK[43078] := 16#9F56;
   // UNICODE_TO_GBK[43079] := 16#FD5C;
   // UNICODE_TO_GBK[43080] := 16#9F57;
   // UNICODE_TO_GBK[43081] := 16#FD5D;
   // UNICODE_TO_GBK[43082] := 16#9F58;
   // UNICODE_TO_GBK[43083] := 16#FD5E;
   // UNICODE_TO_GBK[43084] := 16#9F59;
   // UNICODE_TO_GBK[43085] := 16#FD5F;
   // UNICODE_TO_GBK[43086] := 16#9F5A;
   // UNICODE_TO_GBK[43087] := 16#FD60;
   // UNICODE_TO_GBK[43088] := 16#9F5B;
   // UNICODE_TO_GBK[43089] := 16#FD61;
   // UNICODE_TO_GBK[43090] := 16#9F5C;
   // UNICODE_TO_GBK[43091] := 16#FD62;
   // UNICODE_TO_GBK[43092] := 16#9F5D;
   // UNICODE_TO_GBK[43093] := 16#FD63;
   // UNICODE_TO_GBK[43094] := 16#9F5E;
   // UNICODE_TO_GBK[43095] := 16#FD64;
   // UNICODE_TO_GBK[43096] := 16#9F5F;
   // UNICODE_TO_GBK[43097] := 16#FD65;
   // UNICODE_TO_GBK[43098] := 16#9F60;
   // UNICODE_TO_GBK[43099] := 16#FD66;
   // UNICODE_TO_GBK[43100] := 16#9F61;
   // UNICODE_TO_GBK[43101] := 16#FD67;
   // UNICODE_TO_GBK[43102] := 16#9F62;
   // UNICODE_TO_GBK[43103] := 16#FD68;
   // UNICODE_TO_GBK[43104] := 16#9F63;
   // UNICODE_TO_GBK[43105] := 16#FD69;
   // UNICODE_TO_GBK[43106] := 16#9F64;
   // UNICODE_TO_GBK[43107] := 16#FD6A;
   // UNICODE_TO_GBK[43108] := 16#9F65;
   // UNICODE_TO_GBK[43109] := 16#FD6B;
   // UNICODE_TO_GBK[43110] := 16#9F66;
   // UNICODE_TO_GBK[43111] := 16#FD6C;
   // UNICODE_TO_GBK[43112] := 16#9F67;
   // UNICODE_TO_GBK[43113] := 16#FD6D;
   // UNICODE_TO_GBK[43114] := 16#9F68;
   // UNICODE_TO_GBK[43115] := 16#FD6E;
   // UNICODE_TO_GBK[43116] := 16#9F69;
   // UNICODE_TO_GBK[43117] := 16#FD6F;
   // UNICODE_TO_GBK[43118] := 16#9F6A;
   // UNICODE_TO_GBK[43119] := 16#FD70;
   // UNICODE_TO_GBK[43120] := 16#9F6B;
   // UNICODE_TO_GBK[43121] := 16#FD71;
   // UNICODE_TO_GBK[43122] := 16#9F6C;
   // UNICODE_TO_GBK[43123] := 16#FD72;
   // UNICODE_TO_GBK[43124] := 16#9F6D;
   // UNICODE_TO_GBK[43125] := 16#FD73;
   // UNICODE_TO_GBK[43126] := 16#9F6E;
   // UNICODE_TO_GBK[43127] := 16#FD74;
   // UNICODE_TO_GBK[43128] := 16#9F6F;
   // UNICODE_TO_GBK[43129] := 16#FD75;
   // UNICODE_TO_GBK[43130] := 16#9F70;
   // UNICODE_TO_GBK[43131] := 16#FD76;
   // UNICODE_TO_GBK[43132] := 16#9F71;
   // UNICODE_TO_GBK[43133] := 16#FD77;
   // UNICODE_TO_GBK[43134] := 16#9F72;
   // UNICODE_TO_GBK[43135] := 16#FD78;
   // UNICODE_TO_GBK[43136] := 16#9F73;
   // UNICODE_TO_GBK[43137] := 16#FD79;
   // UNICODE_TO_GBK[43138] := 16#9F74;
   // UNICODE_TO_GBK[43139] := 16#FD7A;
   // UNICODE_TO_GBK[43140] := 16#9F75;
   // UNICODE_TO_GBK[43141] := 16#FD7B;
   // UNICODE_TO_GBK[43142] := 16#9F76;
   // UNICODE_TO_GBK[43143] := 16#FD7C;
   // UNICODE_TO_GBK[43144] := 16#9F77;
   // UNICODE_TO_GBK[43145] := 16#FD7D;
   // UNICODE_TO_GBK[43146] := 16#9F78;
   // UNICODE_TO_GBK[43147] := 16#FD7E;
   // UNICODE_TO_GBK[43148] := 16#9F79;
   // UNICODE_TO_GBK[43149] := 16#FD80;
   // UNICODE_TO_GBK[43150] := 16#9F7A;
   // UNICODE_TO_GBK[43151] := 16#FD81;
   // UNICODE_TO_GBK[43152] := 16#9F7B;
   // UNICODE_TO_GBK[43153] := 16#FD82;
   // UNICODE_TO_GBK[43154] := 16#9F7C;
   // UNICODE_TO_GBK[43155] := 16#FD83;
   // UNICODE_TO_GBK[43156] := 16#9F7D;
   // UNICODE_TO_GBK[43157] := 16#FD84;
   // UNICODE_TO_GBK[43158] := 16#9F7E;
   // UNICODE_TO_GBK[43159] := 16#FD85;
   // UNICODE_TO_GBK[43160] := 16#9F7F;
   // UNICODE_TO_GBK[43161] := 16#B3DD;
   // UNICODE_TO_GBK[43162] := 16#9F80;
   // UNICODE_TO_GBK[43163] := 16#F6B3;
   // UNICODE_TO_GBK[43164] := 16#9F81;
   // UNICODE_TO_GBK[43165] := 16#FD86;
   // UNICODE_TO_GBK[43166] := 16#9F82;
   // UNICODE_TO_GBK[43167] := 16#FD87;
   // UNICODE_TO_GBK[43168] := 16#9F83;
   // UNICODE_TO_GBK[43169] := 16#F6B4;
   // UNICODE_TO_GBK[43170] := 16#9F84;
   // UNICODE_TO_GBK[43171] := 16#C1E4;
   // UNICODE_TO_GBK[43172] := 16#9F85;
   // UNICODE_TO_GBK[43173] := 16#F6B5;
   // UNICODE_TO_GBK[43174] := 16#9F86;
   // UNICODE_TO_GBK[43175] := 16#F6B6;
   // UNICODE_TO_GBK[43176] := 16#9F87;
   // UNICODE_TO_GBK[43177] := 16#F6B7;
   // UNICODE_TO_GBK[43178] := 16#9F88;
   // UNICODE_TO_GBK[43179] := 16#F6B8;
   // UNICODE_TO_GBK[43180] := 16#9F89;
   // UNICODE_TO_GBK[43181] := 16#F6B9;
   // UNICODE_TO_GBK[43182] := 16#9F8A;
   // UNICODE_TO_GBK[43183] := 16#F6BA;
   // UNICODE_TO_GBK[43184] := 16#9F8B;
   // UNICODE_TO_GBK[43185] := 16#C8A3;
   // UNICODE_TO_GBK[43186] := 16#9F8C;
   // UNICODE_TO_GBK[43187] := 16#F6BB;
   // UNICODE_TO_GBK[43188] := 16#9F8D;
   // UNICODE_TO_GBK[43189] := 16#FD88;
   // UNICODE_TO_GBK[43190] := 16#9F8E;
   // UNICODE_TO_GBK[43191] := 16#FD89;
   // UNICODE_TO_GBK[43192] := 16#9F8F;
   // UNICODE_TO_GBK[43193] := 16#FD8A;
   // UNICODE_TO_GBK[43194] := 16#9F90;
   // UNICODE_TO_GBK[43195] := 16#FD8B;
   // UNICODE_TO_GBK[43196] := 16#9F91;
   // UNICODE_TO_GBK[43197] := 16#FD8C;
   // UNICODE_TO_GBK[43198] := 16#9F92;
   // UNICODE_TO_GBK[43199] := 16#FD8D;
   // UNICODE_TO_GBK[43200] := 16#9F93;
   // UNICODE_TO_GBK[43201] := 16#FD8E;
   // UNICODE_TO_GBK[43202] := 16#9F94;
   // UNICODE_TO_GBK[43203] := 16#FD8F;
   // UNICODE_TO_GBK[43204] := 16#9F95;
   // UNICODE_TO_GBK[43205] := 16#FD90;
   // UNICODE_TO_GBK[43206] := 16#9F96;
   // UNICODE_TO_GBK[43207] := 16#FD91;
   // UNICODE_TO_GBK[43208] := 16#9F97;
   // UNICODE_TO_GBK[43209] := 16#FD92;
   // UNICODE_TO_GBK[43210] := 16#9F98;
   // UNICODE_TO_GBK[43211] := 16#FD93;
   // UNICODE_TO_GBK[43212] := 16#9F99;
   // UNICODE_TO_GBK[43213] := 16#C1FA;
   // UNICODE_TO_GBK[43214] := 16#9F9A;
   // UNICODE_TO_GBK[43215] := 16#B9A8;
   // UNICODE_TO_GBK[43216] := 16#9F9B;
   // UNICODE_TO_GBK[43217] := 16#EDE8;
   // UNICODE_TO_GBK[43218] := 16#9F9C;
   // UNICODE_TO_GBK[43219] := 16#FD94;
   // UNICODE_TO_GBK[43220] := 16#9F9D;
   // UNICODE_TO_GBK[43221] := 16#FD95;
   // UNICODE_TO_GBK[43222] := 16#9F9E;
   // UNICODE_TO_GBK[43223] := 16#FD96;
   // UNICODE_TO_GBK[43224] := 16#9F9F;
   // UNICODE_TO_GBK[43225] := 16#B9EA;
   // UNICODE_TO_GBK[43226] := 16#9FA0;
   // UNICODE_TO_GBK[43227] := 16#D9DF;
   // UNICODE_TO_GBK[43228] := 16#9FA1;
   // UNICODE_TO_GBK[43229] := 16#FD97;
   // UNICODE_TO_GBK[43230] := 16#9FA2;
   // UNICODE_TO_GBK[43231] := 16#FD98;
   // UNICODE_TO_GBK[43232] := 16#9FA3;
   // UNICODE_TO_GBK[43233] := 16#FD99;
   // UNICODE_TO_GBK[43234] := 16#9FA4;
   // UNICODE_TO_GBK[43235] := 16#FD9A;
   // UNICODE_TO_GBK[43236] := 16#9FA5;
   // UNICODE_TO_GBK[43237] := 16#FD9B;
   // UNICODE_TO_GBK[43238] := 16#F92C;
   // UNICODE_TO_GBK[43239] := 16#FD9C;
   // UNICODE_TO_GBK[43240] := 16#F979;
   // UNICODE_TO_GBK[43241] := 16#FD9D;
   // UNICODE_TO_GBK[43242] := 16#F995;
   // UNICODE_TO_GBK[43243] := 16#FD9E;
   // UNICODE_TO_GBK[43244] := 16#F9E7;
   // UNICODE_TO_GBK[43245] := 16#FD9F;
   // UNICODE_TO_GBK[43246] := 16#F9F1;
   // UNICODE_TO_GBK[43247] := 16#FDA0;
   // UNICODE_TO_GBK[43248] := 16#FA0C;
   // UNICODE_TO_GBK[43249] := 16#FE40;
   // UNICODE_TO_GBK[43250] := 16#FA0D;
   // UNICODE_TO_GBK[43251] := 16#FE41;
   // UNICODE_TO_GBK[43252] := 16#FA0E;
   // UNICODE_TO_GBK[43253] := 16#FE42;
   // UNICODE_TO_GBK[43254] := 16#FA0F;
   // UNICODE_TO_GBK[43255] := 16#FE43;
   // UNICODE_TO_GBK[43256] := 16#FA11;
   // UNICODE_TO_GBK[43257] := 16#FE44;
   // UNICODE_TO_GBK[43258] := 16#FA13;
   // UNICODE_TO_GBK[43259] := 16#FE45;
   // UNICODE_TO_GBK[43260] := 16#FA14;
   // UNICODE_TO_GBK[43261] := 16#FE46;
   // UNICODE_TO_GBK[43262] := 16#FA18;
   // UNICODE_TO_GBK[43263] := 16#FE47;
   // UNICODE_TO_GBK[43264] := 16#FA1F;
   // UNICODE_TO_GBK[43265] := 16#FE48;
   // UNICODE_TO_GBK[43266] := 16#FA20;
   // UNICODE_TO_GBK[43267] := 16#FE49;
   // UNICODE_TO_GBK[43268] := 16#FA21;
   // UNICODE_TO_GBK[43269] := 16#FE4A;
   // UNICODE_TO_GBK[43270] := 16#FA23;
   // UNICODE_TO_GBK[43271] := 16#FE4B;
   // UNICODE_TO_GBK[43272] := 16#FA24;
   // UNICODE_TO_GBK[43273] := 16#FE4C;
   // UNICODE_TO_GBK[43274] := 16#FA27;
   // UNICODE_TO_GBK[43275] := 16#FE4D;
   // UNICODE_TO_GBK[43276] := 16#FA28;
   // UNICODE_TO_GBK[43277] := 16#FE4E;
   // UNICODE_TO_GBK[43278] := 16#FA29;
   // UNICODE_TO_GBK[43279] := 16#FE4F;
   // UNICODE_TO_GBK[43280] := 16#FE30;
   // UNICODE_TO_GBK[43281] := 16#A955;
   // UNICODE_TO_GBK[43282] := 16#FE31;
   // UNICODE_TO_GBK[43283] := 16#A6F2;
   // UNICODE_TO_GBK[43284] := 16#FE33;
   // UNICODE_TO_GBK[43285] := 16#A6F4;
   // UNICODE_TO_GBK[43286] := 16#FE34;
   // UNICODE_TO_GBK[43287] := 16#A6F5;
   // UNICODE_TO_GBK[43288] := 16#FE35;
   // UNICODE_TO_GBK[43289] := 16#A6E0;
   // UNICODE_TO_GBK[43290] := 16#FE36;
   // UNICODE_TO_GBK[43291] := 16#A6E1;
   // UNICODE_TO_GBK[43292] := 16#FE37;
   // UNICODE_TO_GBK[43293] := 16#A6F0;
   // UNICODE_TO_GBK[43294] := 16#FE38;
   // UNICODE_TO_GBK[43295] := 16#A6F1;
   // UNICODE_TO_GBK[43296] := 16#FE39;
   // UNICODE_TO_GBK[43297] := 16#A6E2;
   // UNICODE_TO_GBK[43298] := 16#FE3A;
   // UNICODE_TO_GBK[43299] := 16#A6E3;
   // UNICODE_TO_GBK[43300] := 16#FE3B;
   // UNICODE_TO_GBK[43301] := 16#A6EE;
   // UNICODE_TO_GBK[43302] := 16#FE3C;
   // UNICODE_TO_GBK[43303] := 16#A6EF;
   // UNICODE_TO_GBK[43304] := 16#FE3D;
   // UNICODE_TO_GBK[43305] := 16#A6E6;
   // UNICODE_TO_GBK[43306] := 16#FE3E;
   // UNICODE_TO_GBK[43307] := 16#A6E7;
   // UNICODE_TO_GBK[43308] := 16#FE3F;
   // UNICODE_TO_GBK[43309] := 16#A6E4;
   // UNICODE_TO_GBK[43310] := 16#FE40;
   // UNICODE_TO_GBK[43311] := 16#A6E5;
   // UNICODE_TO_GBK[43312] := 16#FE41;
   // UNICODE_TO_GBK[43313] := 16#A6E8;
   // UNICODE_TO_GBK[43314] := 16#FE42;
   // UNICODE_TO_GBK[43315] := 16#A6E9;
   // UNICODE_TO_GBK[43316] := 16#FE43;
   // UNICODE_TO_GBK[43317] := 16#A6EA;
   // UNICODE_TO_GBK[43318] := 16#FE44;
   // UNICODE_TO_GBK[43319] := 16#A6EB;
   // UNICODE_TO_GBK[43320] := 16#FE49;
   // UNICODE_TO_GBK[43321] := 16#A968;
   // UNICODE_TO_GBK[43322] := 16#FE4A;
   // UNICODE_TO_GBK[43323] := 16#A969;
   // UNICODE_TO_GBK[43324] := 16#FE4B;
   // UNICODE_TO_GBK[43325] := 16#A96A;
   // UNICODE_TO_GBK[43326] := 16#FE4C;
   // UNICODE_TO_GBK[43327] := 16#A96B;
   // UNICODE_TO_GBK[43328] := 16#FE4D;
   // UNICODE_TO_GBK[43329] := 16#A96C;
   // UNICODE_TO_GBK[43330] := 16#FE4E;
   // UNICODE_TO_GBK[43331] := 16#A96D;
   // UNICODE_TO_GBK[43332] := 16#FE4F;
   // UNICODE_TO_GBK[43333] := 16#A96E;
   // UNICODE_TO_GBK[43334] := 16#FE50;
   // UNICODE_TO_GBK[43335] := 16#A96F;
   // UNICODE_TO_GBK[43336] := 16#FE51;
   // UNICODE_TO_GBK[43337] := 16#A970;
   // UNICODE_TO_GBK[43338] := 16#FE52;
   // UNICODE_TO_GBK[43339] := 16#A971;
   // UNICODE_TO_GBK[43340] := 16#FE54;
   // UNICODE_TO_GBK[43341] := 16#A972;
   // UNICODE_TO_GBK[43342] := 16#FE55;
   // UNICODE_TO_GBK[43343] := 16#A973;
   // UNICODE_TO_GBK[43344] := 16#FE56;
   // UNICODE_TO_GBK[43345] := 16#A974;
   // UNICODE_TO_GBK[43346] := 16#FE57;
   // UNICODE_TO_GBK[43347] := 16#A975;
   // UNICODE_TO_GBK[43348] := 16#FE59;
   // UNICODE_TO_GBK[43349] := 16#A976;
   // UNICODE_TO_GBK[43350] := 16#FE5A;
   // UNICODE_TO_GBK[43351] := 16#A977;
   // UNICODE_TO_GBK[43352] := 16#FE5B;
   // UNICODE_TO_GBK[43353] := 16#A978;
   // UNICODE_TO_GBK[43354] := 16#FE5C;
   // UNICODE_TO_GBK[43355] := 16#A979;
   // UNICODE_TO_GBK[43356] := 16#FE5D;
   // UNICODE_TO_GBK[43357] := 16#A97A;
   // UNICODE_TO_GBK[43358] := 16#FE5E;
   // UNICODE_TO_GBK[43359] := 16#A97B;
   // UNICODE_TO_GBK[43360] := 16#FE5F;
   // UNICODE_TO_GBK[43361] := 16#A97C;
   // UNICODE_TO_GBK[43362] := 16#FE60;
   // UNICODE_TO_GBK[43363] := 16#A97D;
   // UNICODE_TO_GBK[43364] := 16#FE61;
   // UNICODE_TO_GBK[43365] := 16#A97E;
   // UNICODE_TO_GBK[43366] := 16#FE62;
   // UNICODE_TO_GBK[43367] := 16#A980;
   // UNICODE_TO_GBK[43368] := 16#FE63;
   // UNICODE_TO_GBK[43369] := 16#A981;
   // UNICODE_TO_GBK[43370] := 16#FE64;
   // UNICODE_TO_GBK[43371] := 16#A982;
   // UNICODE_TO_GBK[43372] := 16#FE65;
   // UNICODE_TO_GBK[43373] := 16#A983;
   // UNICODE_TO_GBK[43374] := 16#FE66;
   // UNICODE_TO_GBK[43375] := 16#A984;
   // UNICODE_TO_GBK[43376] := 16#FE68;
   // UNICODE_TO_GBK[43377] := 16#A985;
   // UNICODE_TO_GBK[43378] := 16#FE69;
   // UNICODE_TO_GBK[43379] := 16#A986;
   // UNICODE_TO_GBK[43380] := 16#FE6A;
   // UNICODE_TO_GBK[43381] := 16#A987;
   // UNICODE_TO_GBK[43382] := 16#FE6B;
   // UNICODE_TO_GBK[43383] := 16#A988;
   // UNICODE_TO_GBK[43384] := 16#FF01;
   // UNICODE_TO_GBK[43385] := 16#A3A1;
   // UNICODE_TO_GBK[43386] := 16#FF02;
   // UNICODE_TO_GBK[43387] := 16#A3A2;
   // UNICODE_TO_GBK[43388] := 16#FF03;
   // UNICODE_TO_GBK[43389] := 16#A3A3;
   // UNICODE_TO_GBK[43390] := 16#FF04;
   // UNICODE_TO_GBK[43391] := 16#A1E7;
   // UNICODE_TO_GBK[43392] := 16#FF05;
   // UNICODE_TO_GBK[43393] := 16#A3A5;
   // UNICODE_TO_GBK[43394] := 16#FF06;
   // UNICODE_TO_GBK[43395] := 16#A3A6;
   // UNICODE_TO_GBK[43396] := 16#FF07;
   // UNICODE_TO_GBK[43397] := 16#A3A7;
   // UNICODE_TO_GBK[43398] := 16#FF08;
   // UNICODE_TO_GBK[43399] := 16#A3A8;
   // UNICODE_TO_GBK[43400] := 16#FF09;
   // UNICODE_TO_GBK[43401] := 16#A3A9;
   // UNICODE_TO_GBK[43402] := 16#FF0A;
   // UNICODE_TO_GBK[43403] := 16#A3AA;
   // UNICODE_TO_GBK[43404] := 16#FF0B;
   // UNICODE_TO_GBK[43405] := 16#A3AB;
   // UNICODE_TO_GBK[43406] := 16#FF0C;
   // UNICODE_TO_GBK[43407] := 16#A3AC;
   // UNICODE_TO_GBK[43408] := 16#FF0D;
   // UNICODE_TO_GBK[43409] := 16#A3AD;
   // UNICODE_TO_GBK[43410] := 16#FF0E;
   // UNICODE_TO_GBK[43411] := 16#A3AE;
   // UNICODE_TO_GBK[43412] := 16#FF0F;
   // UNICODE_TO_GBK[43413] := 16#A3AF;
   // UNICODE_TO_GBK[43414] := 16#FF10;
   // UNICODE_TO_GBK[43415] := 16#A3B0;
   // UNICODE_TO_GBK[43416] := 16#FF11;
   // UNICODE_TO_GBK[43417] := 16#A3B1;
   // UNICODE_TO_GBK[43418] := 16#FF12;
   // UNICODE_TO_GBK[43419] := 16#A3B2;
   // UNICODE_TO_GBK[43420] := 16#FF13;
   // UNICODE_TO_GBK[43421] := 16#A3B3;
   // UNICODE_TO_GBK[43422] := 16#FF14;
   // UNICODE_TO_GBK[43423] := 16#A3B4;
   // UNICODE_TO_GBK[43424] := 16#FF15;
   // UNICODE_TO_GBK[43425] := 16#A3B5;
   // UNICODE_TO_GBK[43426] := 16#FF16;
   // UNICODE_TO_GBK[43427] := 16#A3B6;
   // UNICODE_TO_GBK[43428] := 16#FF17;
   // UNICODE_TO_GBK[43429] := 16#A3B7;
   // UNICODE_TO_GBK[43430] := 16#FF18;
   // UNICODE_TO_GBK[43431] := 16#A3B8;
   // UNICODE_TO_GBK[43432] := 16#FF19;
   // UNICODE_TO_GBK[43433] := 16#A3B9;
   // UNICODE_TO_GBK[43434] := 16#FF1A;
   // UNICODE_TO_GBK[43435] := 16#A3BA;
   // UNICODE_TO_GBK[43436] := 16#FF1B;
   // UNICODE_TO_GBK[43437] := 16#A3BB;
   // UNICODE_TO_GBK[43438] := 16#FF1C;
   // UNICODE_TO_GBK[43439] := 16#A3BC;
   // UNICODE_TO_GBK[43440] := 16#FF1D;
   // UNICODE_TO_GBK[43441] := 16#A3BD;
   // UNICODE_TO_GBK[43442] := 16#FF1E;
   // UNICODE_TO_GBK[43443] := 16#A3BE;
   // UNICODE_TO_GBK[43444] := 16#FF1F;
   // UNICODE_TO_GBK[43445] := 16#A3BF;
   // UNICODE_TO_GBK[43446] := 16#FF20;
   // UNICODE_TO_GBK[43447] := 16#A3C0;
   // UNICODE_TO_GBK[43448] := 16#FF21;
   // UNICODE_TO_GBK[43449] := 16#A3C1;
   // UNICODE_TO_GBK[43450] := 16#FF22;
   // UNICODE_TO_GBK[43451] := 16#A3C2;
   // UNICODE_TO_GBK[43452] := 16#FF23;
   // UNICODE_TO_GBK[43453] := 16#A3C3;
   // UNICODE_TO_GBK[43454] := 16#FF24;
   // UNICODE_TO_GBK[43455] := 16#A3C4;
   // UNICODE_TO_GBK[43456] := 16#FF25;
   // UNICODE_TO_GBK[43457] := 16#A3C5;
   // UNICODE_TO_GBK[43458] := 16#FF26;
   // UNICODE_TO_GBK[43459] := 16#A3C6;
   // UNICODE_TO_GBK[43460] := 16#FF27;
   // UNICODE_TO_GBK[43461] := 16#A3C7;
   // UNICODE_TO_GBK[43462] := 16#FF28;
   // UNICODE_TO_GBK[43463] := 16#A3C8;
   // UNICODE_TO_GBK[43464] := 16#FF29;
   // UNICODE_TO_GBK[43465] := 16#A3C9;
   // UNICODE_TO_GBK[43466] := 16#FF2A;
   // UNICODE_TO_GBK[43467] := 16#A3CA;
   // UNICODE_TO_GBK[43468] := 16#FF2B;
   // UNICODE_TO_GBK[43469] := 16#A3CB;
   // UNICODE_TO_GBK[43470] := 16#FF2C;
   // UNICODE_TO_GBK[43471] := 16#A3CC;
   // UNICODE_TO_GBK[43472] := 16#FF2D;
   // UNICODE_TO_GBK[43473] := 16#A3CD;
   // UNICODE_TO_GBK[43474] := 16#FF2E;
   // UNICODE_TO_GBK[43475] := 16#A3CE;
   // UNICODE_TO_GBK[43476] := 16#FF2F;
   // UNICODE_TO_GBK[43477] := 16#A3CF;
   // UNICODE_TO_GBK[43478] := 16#FF30;
   // UNICODE_TO_GBK[43479] := 16#A3D0;
   // UNICODE_TO_GBK[43480] := 16#FF31;
   // UNICODE_TO_GBK[43481] := 16#A3D1;
   // UNICODE_TO_GBK[43482] := 16#FF32;
   // UNICODE_TO_GBK[43483] := 16#A3D2;
   // UNICODE_TO_GBK[43484] := 16#FF33;
   // UNICODE_TO_GBK[43485] := 16#A3D3;
   // UNICODE_TO_GBK[43486] := 16#FF34;
   // UNICODE_TO_GBK[43487] := 16#A3D4;
   // UNICODE_TO_GBK[43488] := 16#FF35;
   // UNICODE_TO_GBK[43489] := 16#A3D5;
   // UNICODE_TO_GBK[43490] := 16#FF36;
   // UNICODE_TO_GBK[43491] := 16#A3D6;
   // UNICODE_TO_GBK[43492] := 16#FF37;
   // UNICODE_TO_GBK[43493] := 16#A3D7;
   // UNICODE_TO_GBK[43494] := 16#FF38;
   // UNICODE_TO_GBK[43495] := 16#A3D8;
   // UNICODE_TO_GBK[43496] := 16#FF39;
   // UNICODE_TO_GBK[43497] := 16#A3D9;
   // UNICODE_TO_GBK[43498] := 16#FF3A;
   // UNICODE_TO_GBK[43499] := 16#A3DA;
   // UNICODE_TO_GBK[43500] := 16#FF3B;
   // UNICODE_TO_GBK[43501] := 16#A3DB;
   // UNICODE_TO_GBK[43502] := 16#FF3C;
   // UNICODE_TO_GBK[43503] := 16#A3DC;
   // UNICODE_TO_GBK[43504] := 16#FF3D;
   // UNICODE_TO_GBK[43505] := 16#A3DD;
   // UNICODE_TO_GBK[43506] := 16#FF3E;
   // UNICODE_TO_GBK[43507] := 16#A3DE;
   // UNICODE_TO_GBK[43508] := 16#FF3F;
   // UNICODE_TO_GBK[43509] := 16#A3DF;
   // UNICODE_TO_GBK[43510] := 16#FF40;
   // UNICODE_TO_GBK[43511] := 16#A3E0;
   // UNICODE_TO_GBK[43512] := 16#FF41;
   // UNICODE_TO_GBK[43513] := 16#A3E1;
   // UNICODE_TO_GBK[43514] := 16#FF42;
   // UNICODE_TO_GBK[43515] := 16#A3E2;
   // UNICODE_TO_GBK[43516] := 16#FF43;
   // UNICODE_TO_GBK[43517] := 16#A3E3;
   // UNICODE_TO_GBK[43518] := 16#FF44;
   // UNICODE_TO_GBK[43519] := 16#A3E4;
   // UNICODE_TO_GBK[43520] := 16#FF45;
   // UNICODE_TO_GBK[43521] := 16#A3E5;
   // UNICODE_TO_GBK[43522] := 16#FF46;
   // UNICODE_TO_GBK[43523] := 16#A3E6;
   // UNICODE_TO_GBK[43524] := 16#FF47;
   // UNICODE_TO_GBK[43525] := 16#A3E7;
   // UNICODE_TO_GBK[43526] := 16#FF48;
   // UNICODE_TO_GBK[43527] := 16#A3E8;
   // UNICODE_TO_GBK[43528] := 16#FF49;
   // UNICODE_TO_GBK[43529] := 16#A3E9;
   // UNICODE_TO_GBK[43530] := 16#FF4A;
   // UNICODE_TO_GBK[43531] := 16#A3EA;
   // UNICODE_TO_GBK[43532] := 16#FF4B;
   // UNICODE_TO_GBK[43533] := 16#A3EB;
   // UNICODE_TO_GBK[43534] := 16#FF4C;
   // UNICODE_TO_GBK[43535] := 16#A3EC;
   // UNICODE_TO_GBK[43536] := 16#FF4D;
   // UNICODE_TO_GBK[43537] := 16#A3ED;
   // UNICODE_TO_GBK[43538] := 16#FF4E;
   // UNICODE_TO_GBK[43539] := 16#A3EE;
   // UNICODE_TO_GBK[43540] := 16#FF4F;
   // UNICODE_TO_GBK[43541] := 16#A3EF;
   // UNICODE_TO_GBK[43542] := 16#FF50;
   // UNICODE_TO_GBK[43543] := 16#A3F0;
   // UNICODE_TO_GBK[43544] := 16#FF51;
   // UNICODE_TO_GBK[43545] := 16#A3F1;
   // UNICODE_TO_GBK[43546] := 16#FF52;
   // UNICODE_TO_GBK[43547] := 16#A3F2;
   // UNICODE_TO_GBK[43548] := 16#FF53;
   // UNICODE_TO_GBK[43549] := 16#A3F3;
   // UNICODE_TO_GBK[43550] := 16#FF54;
   // UNICODE_TO_GBK[43551] := 16#A3F4;
   // UNICODE_TO_GBK[43552] := 16#FF55;
   // UNICODE_TO_GBK[43553] := 16#A3F5;
   // UNICODE_TO_GBK[43554] := 16#FF56;
   // UNICODE_TO_GBK[43555] := 16#A3F6;
   // UNICODE_TO_GBK[43556] := 16#FF57;
   // UNICODE_TO_GBK[43557] := 16#A3F7;
   // UNICODE_TO_GBK[43558] := 16#FF58;
   // UNICODE_TO_GBK[43559] := 16#A3F8;
   // UNICODE_TO_GBK[43560] := 16#FF59;
   // UNICODE_TO_GBK[43561] := 16#A3F9;
   // UNICODE_TO_GBK[43562] := 16#FF5A;
   // UNICODE_TO_GBK[43563] := 16#A3FA;
   // UNICODE_TO_GBK[43564] := 16#FF5B;
   // UNICODE_TO_GBK[43565] := 16#A3FB;
   // UNICODE_TO_GBK[43566] := 16#FF5C;
   // UNICODE_TO_GBK[43567] := 16#A3FC;
   // UNICODE_TO_GBK[43568] := 16#FF5D;
   // UNICODE_TO_GBK[43569] := 16#A3FD;
   // UNICODE_TO_GBK[43570] := 16#FF5E;
   // UNICODE_TO_GBK[43571] := 16#A1AB;
   // UNICODE_TO_GBK[43572] := 16#FFE0;
   // UNICODE_TO_GBK[43573] := 16#A1E9;
   // UNICODE_TO_GBK[43574] := 16#FFE1;
   // UNICODE_TO_GBK[43575] := 16#A1EA;
   // UNICODE_TO_GBK[43576] := 16#FFE2;
   // UNICODE_TO_GBK[43577] := 16#A956;
   // UNICODE_TO_GBK[43578] := 16#FFE3;
   // UNICODE_TO_GBK[43579] := 16#A3FE;
   // UNICODE_TO_GBK[43580] := 16#FFE4;
   // UNICODE_TO_GBK[43581] := 16#A957;
   // UNICODE_TO_GBK[43582] := 16#FFE5;
   // UNICODE_TO_GBK[43583] := 16#A3A4;
   // UNICODE_TO_GBK[43584] := 0;
   // UNICODE_TO_GBK[43585] := 0;
BEGIN
   IF #UNICODE < 16#0080 THEN
       #GBK := #UNICODE;
   ELSE
       #hi := 21796;
       #li := 0;
       FOR #j := 0 TO 16 BY 1 DO
           #i := #li + (#hi - #li) / 2;
           IF #UNICODE = #UNICODE_TO_GBK[#i * 2] THEN
               #GBK := #UNICODE_TO_GBK[#i * 2 + 1];
               EXIT;
           END_IF;
           IF #UNICODE > #UNICODE_TO_GBK[#i * 2] THEN
               #li := #i;
           ELSE
               #hi := #i;
           END_IF;
       END_FOR;
   END_IF;
END_FUNCTION_BLOCK

// ===== library: MasterCopy "UNI_TO_UTF8" =====

// folder: FB/UNICODE_FB

FUNCTION_BLOCK "UNI_TO_UTF8"   // FB3, SCL
{ S7_Optimized_Access := 'TRUE' }
VERSION : 0.1
   VAR_INPUT
      UNICODE : Word;
   END_VAR
   VAR_OUTPUT
      UTF8 : String[4];
   END_VAR
   VAR_TEMP
      TempStr : String[4];
   END_VAR
BEGIN
   #TempStr := '0000';
   IF #UNICODE <= 16#0000007F THEN
       #TempStr[1] := WORD_TO_BYTE(#UNICODE AND 16#7F);//0111 1111
       #UTF8 := LEFT(IN := #TempStr, L := 1);
   ELSIF #UNICODE > 16#00000080 AND #UNICODE <= 16#000007FF THEN
       #TempStr[2] := WORD_TO_BYTE((#UNICODE AND 16#3F) OR 16#80);//0111 1111            1000 0000
       #TempStr[1] := WORD_TO_BYTE((SHR(IN := #UNICODE, N := 6) AND 16#1F) OR 16#C0);//0001 1111     1100 0000
       #UTF8 := LEFT(IN := #TempStr, L := 2);
   ELSIF #UNICODE > 16#00000800 AND #UNICODE <= 16#0000FFFF THEN
       #TempStr[3] := WORD_TO_BYTE((#UNICODE AND 16#3F) OR 16#80);
       #TempStr[2] := WORD_TO_BYTE((SHR(IN := #UNICODE, N := 6) AND 16#3F) OR 16#80);
       #TempStr[1] := WORD_TO_BYTE((SHR(IN := #UNICODE, N := 12) AND 16#0F) OR 16#E0);
       #UTF8 := LEFT(IN := #TempStr, L := 3);
   END_IF;
END_FUNCTION_BLOCK

// ===== library: MasterCopy "UTF8_TO_UNI" =====

// folder: FB/UNICODE_FB

FUNCTION_BLOCK "UTF8_TO_UNI"   // FB4, SCL
{ S7_Optimized_Access := 'TRUE' }
VERSION : 0.1
   VAR_INPUT
      UTF8 : String[4];
   END_VAR
   VAR_OUTPUT
      UNICODE : Word;
   END_VAR
   VAR_TEMP
      TempDW : DWord;
      TempW : Array[0..3] of Word;
   END_VAR
BEGIN
   #TempDW := #UTF8[1];
   IF #TempDW < 16#80 THEN
       #UNICODE := DWORD_TO_WORD(#TempDW AND 16#7F);
   ELSIF #TempDW >= 16#80 AND #TempDW < 16#C0 THEN
       ;
   ELSIF #TempDW >= 16#C0 AND #TempDW < 16#E0 THEN
       #TempDW := SHL(IN := #TempDW, N := 8);
       #TempDW := #TempDW + BYTE_TO_WORD(#UTF8[2]);
       #TempW[0] := DWORD_TO_WORD(SHR(IN:=#TempDW AND 16#1F00, N:=2));
       #TempW[1] := DWORD_TO_WORD(#TempDW AND 16#3F);
       #UNICODE := #TempW[0] + #TempW[1];
   ELSIF #TempDW >= 16#E0 AND #TempDW < 16#F0 THEN
       #TempDW := SHL(IN := #TempDW, N := 8);
       #TempDW := #TempDW + BYTE_TO_WORD(#UTF8[2]);
       #TempDW := SHL(IN := #TempDW, N := 8);
       #TempDW := #TempDW + BYTE_TO_WORD(#UTF8[3]);
       #TempW[0] := DWORD_TO_WORD(SHR(IN:=#TempDW AND 16#0F0000, N:=4));
       #TempW[1] := DWORD_TO_WORD(SHR(IN:=#TempDW AND 16#3F00, N:=2));
       #TempW[2] := DWORD_TO_WORD(#TempDW AND 16#3F);
       #UNICODE := #TempW[0] + #TempW[1] + #TempW[2];
   ELSIF #TempDW >= 16#F0 AND #TempDW < 16#F8 THEN
       #TempDW := SHL(IN := #TempDW,  N := 8);
       #TempDW := #TempDW + BYTE_TO_WORD(#UTF8[2]);
       #TempDW := SHL(IN := #TempDW, N := 8);
       #TempDW := #TempDW + BYTE_TO_WORD(#UTF8[3]);
       #TempDW := SHL(IN := #TempDW,  N := 8);
       #TempDW := #TempDW + BYTE_TO_WORD(#UTF8[4]);
       #TempW[0] := DWORD_TO_WORD(SHR(IN:=#TempDW AND 16#7000000, N:=6));
       #TempW[1] := DWORD_TO_WORD(SHR(IN:=#TempDW AND 16#3F0000, N:=4));
       #TempW[2] := DWORD_TO_WORD(SHR(IN:=#TempDW AND 16#3F00, N:=2));
       #TempW[3] := DWORD_TO_WORD(#TempDW AND 16#3F);
       #UNICODE := #TempW[0] + #TempW[1] + #TempW[2] + #TempW[3];
   END_IF;
END_FUNCTION_BLOCK

// ===== library: MasterCopy "喷码机01追加数据" =====

// folder: FC/喷码机

FUNCTION "喷码机01追加数据" : String   // FC1, SCL
{ S7_Optimized_Access := 'TRUE' }
VERSION : 0.1
   VAR_INPUT
      X0信息 : String;
      X1信息 : String;
      X2信息 : String;
      X3信息 : String;
   END_VAR
   VAR_TEMP
      X0长度 : Int;
      X1长度 : Int;
      X2长度 : Int;
      X3长度 : Int;
      转换信息 : String;
      i : Int;
      j : DInt;
      Temp_Str : String;
      求和 : DWord;
      Checksum : Word;
      Temp_Chars : Array[1..250] of Byte;
   END_VAR
BEGIN
   #X0长度 := LEN(#X0信息);
   #X1长度 := LEN(#X1信息);
   #X2长度 := LEN(#X2信息);
   #X3长度 := LEN(#X3信息);
   IF #X0长度>0 OR #X1长度>0 OR #X2长度>0 OR #X3长度>0 THEN
       #转换信息 := '';
       IF #X0长度 > 0 THEN                                      //X0
           #转换信息 := CONCAT(IN1 := #转换信息,IN2 :=  '00580030');
           Strg_TO_Chars(Strg := #X0信息,
                         pChars := 0,
                         Cnt =>  #j,
                         Chars := #Temp_Chars);
           FOR #i := 1 TO #X0长度 BY 1 DO               //信息X0内容转为明码
               #j := HTA(IN := #Temp_Chars[#i], N := 1, OUT => #Temp_Str);
               IF #Temp_Chars[#i] < 128 THEN
                   #Temp_Str := CONCAT(IN1 := '00', IN2 := #Temp_Str);
               END_IF;
               #转换信息 := CONCAT(IN1 := #转换信息, IN2 := #Temp_Str);
           END_FOR;
           #转换信息 := CONCAT(IN1 := #转换信息,IN2 :=  '001F');
       END_IF;//.............................................................
       IF #X1长度 > 0 THEN                                      //X1
           #转换信息 := CONCAT(IN1 := #转换信息, IN2 := '00580031');
           Strg_TO_Chars(Strg := #X1信息,
                         pChars := 0,
                         Cnt => #j,
                         Chars := #Temp_Chars);
           FOR #i := 1 TO #X1长度 BY 1 DO               //信息X1内容转为明码
               #j := HTA(IN := #Temp_Chars[#i], N := 1, OUT => #Temp_Str);
               IF #Temp_Chars[#i] < 128 THEN
                   #Temp_Str := CONCAT(IN1 := '00', IN2 := #Temp_Str);
               END_IF;
               #转换信息 := CONCAT(IN1 := #转换信息, IN2 := #Temp_Str);
           END_FOR;
           #转换信息 := CONCAT(IN1 := #转换信息, IN2 := '001F');
       END_IF;//.............................................................    
       IF #X2长度 > 0 THEN                                      //X2
           #转换信息 := CONCAT(IN1 := #转换信息, IN2 := '00580032');
           Strg_TO_Chars(Strg := #X2信息,
                         pChars := 0,
                         Cnt => #j,
                         Chars := #Temp_Chars);
           FOR #i := 1 TO #X2长度 BY 1 DO               //信息X2内容转为明码
               #j := HTA(IN := #Temp_Chars[#i], N := 1, OUT => #Temp_Str);
               IF #Temp_Chars[#i] < 128 THEN
                   #Temp_Str := CONCAT(IN1 := '00', IN2 := #Temp_Str);
               END_IF;
               #转换信息 := CONCAT(IN1 := #转换信息, IN2 := #Temp_Str);
           END_FOR;
           #转换信息 := CONCAT(IN1 := #转换信息, IN2 := '001F');
       END_IF;//.............................................................
       IF #X3长度 > 0 THEN                                      //X3
           #转换信息 := CONCAT(IN1 := #转换信息, IN2 := '00580033');
           Strg_TO_Chars(Strg := #X3信息,
                         pChars := 0,
                         Cnt => #j,
                         Chars := #Temp_Chars);
           FOR #i := 1 TO #X3长度 BY 1 DO               //信息X3内容转为明码
               #j := HTA(IN := #Temp_Chars[#i], N := 1, OUT => #Temp_Str);
               IF #Temp_Chars[#i] < 128 THEN
                   #Temp_Str := CONCAT(IN1 := '00', IN2 := #Temp_Str);
               END_IF;
               #转换信息 := CONCAT(IN1 := #转换信息, IN2 := #Temp_Str);
           END_FOR;
           #转换信息 := CONCAT(IN1 := #转换信息, IN2 := '001F');
       END_IF;//.............................................................      
       #j := HTA(IN := LEN(#转换信息), N := 4, OUT => #Temp_Str);//Length明码
       #Temp_Str := LEFT(IN := #Temp_Str, L := 4);//for 1500
       #转换信息 := CONCAT(IN1 := #Temp_Str, IN2 := #转换信息);
       #转换信息 := CONCAT(IN1 := '01', IN2 := #转换信息);//
       #转换信息 := CONCAT(IN1 := '01', IN2 := #转换信息);//OrderID    
       #求和 := 0;//.........................................................................
       Strg_TO_Chars(Strg := #转换信息,
                     pChars := 0,
                     Cnt => #j,
                     Chars := #Temp_Chars);
       FOR #i := 1 TO LEN(#转换信息) DO//求和
           #求和 := #求和 + #Temp_Chars[#i];
       END_FOR;//....................................................................................
       #Checksum := DWORD_TO_WORD(#求和 MOD 65536);
       #Checksum := NOT #Checksum;
       #Checksum := #Checksum + 1; //Checksum
       #j := HTA(IN := #Checksum, N := 4, OUT => #Temp_Str);//Checksum明码.....
       #Temp_Str := LEFT(IN := #Temp_Str, L := 4);//for 1500
       #转换信息 := CONCAT(IN1 := #转换信息, IN2 := #Temp_Str);
       #转换信息 := CONCAT(IN1 := '~', IN2 :=  #转换信息);        //起始码
       #转换信息 := CONCAT(IN1 := #转换信息, IN2 :=  '$R');       //结束码
       #喷码机01追加数据 := #转换信息;
   ELSE
       #喷码机01追加数据 := '';
   END_IF;
END_FUNCTION

// ===== library: MasterCopy "HEX_TO_WORD" =====

// folder: FC/喷码机

FUNCTION "HEX_TO_WORD" : Word   // FC9, SCL
{ S7_Optimized_Access := 'TRUE' }
VERSION : 0.1
   VAR_INPUT
      HEX : String;
   END_VAR
   VAR_TEMP
      i : Int;
      X : Byte;
      W : Word;
   END_VAR
BEGIN
   #W := 0;
   FOR #i := 1 TO 4 DO
       #X := #HEX[#i];
       IF #X > 47 AND #X < 58 THEN
           #W := SHL(IN:=#W, N:=4) + #X - 48;
       ELSIF #X > 64 AND #X < 71 THEN
           #W := SHL(IN:=#W, N:=4) + #X - 55;
       ELSIF #X > 96 AND #X < 103 THEN
           #W := SHL(IN:=#W, N:=4) + #X - 87;
       END_IF;
   END_FOR;
   #HEX_TO_WORD := #W;
END_FUNCTION

// ===== library: MasterCopy "喷码机02更新数据" =====

// folder: FC/喷码机

FUNCTION "喷码机02更新数据" : String   // FC2, SCL
{ S7_Optimized_Access := 'TRUE' }
VERSION : 0.1
   VAR_INPUT
      X0信息 : String;
      X1信息 : String;
      X2信息 : String;
      X3信息 : String;
   END_VAR
   VAR_TEMP
      X0长度 : Int;
      X1长度 : Int;
      X2长度 : Int;
      X3长度 : Int;
      转换信息 : String;
      i : Int;
      j : DInt;
      Temp_Str : String;
      求和 : DWord;
      Checksum : Word;
      Temp_Chars : Array[1..250] of Byte;
   END_VAR
BEGIN
   #X0长度 := LEN(#X0信息);
   #X1长度 := LEN(#X1信息);
   #X2长度 := LEN(#X2信息);
   #X3长度 := LEN(#X3信息);
   IF #X0长度>0 OR #X1长度>0 OR #X2长度>0 OR #X3长度>0 THEN
       #转换信息 := '';
       IF #X0长度 > 0 THEN                                      //X0
           #转换信息 := CONCAT(IN1 := #转换信息,IN2 :=  '00580030');
           Strg_TO_Chars(Strg := #X0信息,
                         pChars := 0,
                         Cnt =>  #j,
                         Chars := #Temp_Chars);
           FOR #i := 1 TO #X0长度 BY 1 DO               //信息X0内容转为明码
               #j := HTA(IN := #Temp_Chars[#i], N := 1, OUT => #Temp_Str);
               IF #Temp_Chars[#i] < 128 THEN
                   #Temp_Str := CONCAT(IN1 := '00', IN2 := #Temp_Str);
               END_IF;
               #转换信息 := CONCAT(IN1 := #转换信息, IN2 := #Temp_Str);
           END_FOR;
           #转换信息 := CONCAT(IN1 := #转换信息,IN2 :=  '001F');
       END_IF;//.............................................................
       IF #X1长度 > 0 THEN                                      //X1
           #转换信息 := CONCAT(IN1 := #转换信息, IN2 := '00580031');
           Strg_TO_Chars(Strg := #X1信息,
                         pChars := 0,
                         Cnt => #j,
                         Chars := #Temp_Chars);
           FOR #i := 1 TO #X1长度 BY 1 DO               //信息X1内容转为明码
               #j := HTA(IN := #Temp_Chars[#i], N := 1, OUT => #Temp_Str);
               IF #Temp_Chars[#i] < 128 THEN
                   #Temp_Str := CONCAT(IN1 := '00', IN2 := #Temp_Str);
               END_IF;
               #转换信息 := CONCAT(IN1 := #转换信息, IN2 := #Temp_Str);
           END_FOR;
           #转换信息 := CONCAT(IN1 := #转换信息, IN2 := '001F');
       END_IF;//.............................................................    
       IF #X2长度 > 0 THEN                                      //X2
           #转换信息 := CONCAT(IN1 := #转换信息, IN2 := '00580032');
           Strg_TO_Chars(Strg := #X2信息,
                         pChars := 0,
                         Cnt => #j,
                         Chars := #Temp_Chars);
           FOR #i := 1 TO #X2长度 BY 1 DO               //信息X2内容转为明码
               #j := HTA(IN := #Temp_Chars[#i], N := 1, OUT => #Temp_Str);
               IF #Temp_Chars[#i] < 128 THEN
                   #Temp_Str := CONCAT(IN1 := '00', IN2 := #Temp_Str);
               END_IF;
               #转换信息 := CONCAT(IN1 := #转换信息, IN2 := #Temp_Str);
           END_FOR;
           #转换信息 := CONCAT(IN1 := #转换信息, IN2 := '001F');
       END_IF;//.............................................................
       IF #X3长度 > 0 THEN                                      //X3
           #转换信息 := CONCAT(IN1 := #转换信息, IN2 := '00580033');
           Strg_TO_Chars(Strg := #X3信息,
                         pChars := 0,
                         Cnt => #j,
                         Chars := #Temp_Chars);
           FOR #i := 1 TO #X3长度 BY 1 DO               //信息X3内容转为明码
               #j := HTA(IN := #Temp_Chars[#i], N := 1, OUT => #Temp_Str);
               IF #Temp_Chars[#i] < 128 THEN
                   #Temp_Str := CONCAT(IN1 := '00', IN2 := #Temp_Str);
               END_IF;
               #转换信息 := CONCAT(IN1 := #转换信息, IN2 := #Temp_Str);
           END_FOR;
           #转换信息 := CONCAT(IN1 := #转换信息, IN2 := '001F');
       END_IF;//.............................................................      
       #j := HTA(IN := LEN(#转换信息), N := 4, OUT => #Temp_Str);//Length明码
       #Temp_Str := LEFT(IN := #Temp_Str, L := 4);//for 1500
       #转换信息 := CONCAT(IN1 := #Temp_Str, IN2 := #转换信息);
       #转换信息 := CONCAT(IN1 := '01', IN2 := #转换信息);//追加或更新
       #转换信息 := CONCAT(IN1 := '01', IN2 := #转换信息);//OrderID    
       #求和 := 0;//.........................................................................
       Strg_TO_Chars(Strg := #转换信息,
                     pChars := 0,
                     Cnt => #j,
                     Chars := #Temp_Chars);
       FOR #i := 1 TO LEN(#转换信息) DO//求和
           #求和 := #求和 + #Temp_Chars[#i];
       END_FOR;//....................................................................................
       #Checksum := DWORD_TO_WORD(#求和 MOD 65536);
       #Checksum := NOT #Checksum;
       #Checksum := #Checksum + 1; //Checksum
       #j := HTA(IN := #Checksum, N := 4, OUT => #Temp_Str);//Checksum明码.....
       #Temp_Str := LEFT(IN := #Temp_Str, L := 4);//for 1500
       #转换信息 := CONCAT(IN1 := #转换信息, IN2 := #Temp_Str);
       #转换信息 := CONCAT(IN1 := '~', IN2 :=  #转换信息);        //起始码
       #转换信息 := CONCAT(IN1 := #转换信息, IN2 :=  '$R');       //结束码
       #喷码机02更新数据 := #转换信息;
   ELSE
       #喷码机02更新数据 := '';
   END_IF;
END_FUNCTION

// ===== library: MasterCopy "喷码机03清理用户区" =====

// folder: FC/喷码机

FUNCTION "喷码机03清理用户区" : String   // FC3, SCL
{ S7_Optimized_Access := 'TRUE' }
VERSION : 0.1
   VAR_TEMP
      转换信息 : String;
   END_VAR
BEGIN
   #转换信息 := '03000000FE7D';
   #转换信息 := CONCAT(IN1:='~', IN2:=#转换信息);        //起始码
   #转换信息 := CONCAT(IN1:=#转换信息, IN2:='$R');       //结束码
   #喷码机03清理用户区 := #转换信息;
END_FUNCTION

// ===== library: MasterCopy "喷码机04故障查询" =====

// folder: FC/喷码机

FUNCTION "喷码机04故障查询" : String   // FC4, SCL
{ S7_Optimized_Access := 'TRUE' }
VERSION : 0.1
   VAR_TEMP
      转换信息 : String;
   END_VAR
BEGIN
   #转换信息 := '04000000FE7C';
   #转换信息 := CONCAT(IN1:='~', IN2:=#转换信息);        //起始码
   #转换信息 := CONCAT(IN1:=#转换信息, IN2:='$R');       //结束码
   #喷码机04故障查询 := #转换信息;
END_FUNCTION

// ===== library: MasterCopy "喷码机05开始喷印" =====

// folder: FC/喷码机

FUNCTION "喷码机05开始喷印" : String   // FC5, SCL
{ S7_Optimized_Access := 'TRUE' }
VERSION : 0.1
   VAR_TEMP
      转换信息 : String;
   END_VAR
BEGIN
   #转换信息 := '08000000FE78';
   #转换信息 := CONCAT(IN1:='~', IN2:=#转换信息);        //起始码
   #转换信息 := CONCAT(IN1:=#转换信息, IN2:='$R');       //结束码
   #喷码机05开始喷印 := #转换信息;
END_FUNCTION

// ===== library: MasterCopy "喷码机06结束喷印" =====

// folder: FC/喷码机

FUNCTION "喷码机06结束喷印" : String   // FC6, SCL
{ S7_Optimized_Access := 'TRUE' }
VERSION : 0.1
   VAR_TEMP
      转换信息 : String;
   END_VAR
BEGIN
   #转换信息 := '09000000FE77';
   #转换信息 := CONCAT(IN1:='~', IN2:=#转换信息);        //起始码
   #转换信息 := CONCAT(IN1:=#转换信息, IN2:='$R');       //结束码
   #喷码机06结束喷印 := #转换信息;
END_FUNCTION

// ===== library: MasterCopy "喷码机故障返回" =====

// folder: FC/喷码机

FUNCTION "喷码机故障返回" : Bool   // FC7, SCL
{ S7_Optimized_Access := 'TRUE' }
VERSION : 0.1
   VAR_INPUT
      返回数据 : String;
   END_VAR
   VAR_OUTPUT
      高压故障 : Bool;
      回收信号故障 : Bool;
      机箱温度过高 : Bool;
      混合缸空 : Bool;
      充电故障 : Bool;
      喷头盖打开 : Bool;
      风扇故障 : Bool;
      墨水缸空 : Bool;
      溶剂缸空 : Bool;
      混合缸满 : Bool;
      粘度错误 : Bool;
      粘度检测错误 : Bool;
      同步器过快 : Bool;
   END_VAR
   VAR_TEMP
      OrderID : Byte;
      RTN : Byte;
      BackData : Word;
      CheckSum : String;
      Temp_Str : String;
      求和 : DWord;
      i : UDInt;
      j : UDInt;
      故障信息 : Word;
      Temp_Chars : Array[0..20] of Byte;
      Temp_Word : Word;
      系统故障 : Array[0..15] of Bool;
   END_VAR
BEGIN
   IF LEN(#返回数据) = 14 THEN
       #Temp_Str := MID(IN := #返回数据, L := 2, P := 2);
       #j := ATH(IN := #Temp_Str, N := 2, OUT => #OrderID);
       #Temp_Str := MID(IN := #返回数据, L := 2, P := 4);
       #j := ATH(IN := #Temp_Str, N := 2, OUT => #RTN);
       #Temp_Str := MID(IN := #返回数据, L := 4, P := 6);
       #j := ATH(IN := #Temp_Str, N := 4, OUT => #BackData);
       #CheckSum := MID(IN := #返回数据, L := 4, P := 10);
       #求和 := 0;//..........................................................
       Strg_TO_Chars(Strg := #返回数据,
                     pChars := 0,
                     Cnt => #j,
                     Chars := #Temp_Chars);
       FOR #i := 1 TO 8 BY 1 DO
           #求和 := #求和 + #Temp_Chars[#i];
       END_FOR;
       #Temp_Word := DWORD_TO_WORD(#求和 MOD 65536);
       #Temp_Word := NOT #Temp_Word;
       #Temp_Word := #Temp_Word + 1; //Checksum
       #j := HTA(IN := #Temp_Word, N := 4, OUT => #Temp_Str);//Checksum明码.....
       IF #Temp_Str = #CheckSum THEN
           #喷码机故障返回 := 1;
       ELSE
           #喷码机故障返回 := 0;
       END_IF;
       IF #OrderID = 16#04 OR #OrderID = 16#FE THEN
           #故障信息 := #BackData;
           #Temp_Word := #BackData AND 16#0001;
           FOR #i := 1 TO 16 DO
               IF #Temp_Word <> 0 THEN
                   #系统故障[#i] := 1;
               END_IF;
               #Temp_Word := SHR(IN := #BackData, N := (#i)) AND 16#0001;
           END_FOR;
           #高压故障 := #系统故障[0];
           #回收信号故障 := #系统故障[1];
           #机箱温度过高 := #系统故障[2];
           #混合缸空 := #系统故障[3];
           #充电故障 := #系统故障[4];
           #喷头盖打开 := #系统故障[5];
           #风扇故障 := #系统故障[8];
           #墨水缸空 := #系统故障[9];
           #溶剂缸空 := #系统故障[10];
           #混合缸满 := #系统故障[11];
           #粘度错误 := #系统故障[12];
           #粘度检测错误 := #系统故障[13];
           #同步器过快 := #系统故障[14];
       END_IF;
   ELSE
       #喷码机故障返回 := 0;
   END_IF;
END_FUNCTION

// ===== library: MasterCopy "喷码机数据返回" =====

// folder: FC/喷码机

FUNCTION "喷码机数据返回" : Bool   // FC8, SCL
{ S7_Optimized_Access := 'TRUE' }
VERSION : 0.1
   VAR_INPUT
      返回数据 : String;
   END_VAR
   VAR_OUTPUT
      数据条数 : UInt;
      已满1000条 : Bool;
      不在喷印状态 : Bool;
      上一条信息没有喷完 : Bool;
   END_VAR
   VAR_TEMP
      OrderID : Byte;
      RTN : Byte;
      BackData : Word;
      CheckSum : String;
      Temp_Str : String;
      求和 : DWord;
      i : UDInt;
      j : UDInt;
      Temp_Chars : Array[0..20] of Byte;
      Temp_Word : Word;
   END_VAR
BEGIN
   IF LEN(#返回数据) = 14 THEN
       #Temp_Str := MID(IN := #返回数据, L := 2, P := 2);
       #j := ATH(IN := #Temp_Str, N := 2, OUT => #OrderID);
       #Temp_Str := MID(IN := #返回数据, L := 2, P := 4);
       #j := ATH(IN := #Temp_Str, N := 2, OUT => #RTN);
       #Temp_Str := MID(IN := #返回数据, L := 4, P := 6);
       #j := ATH(IN := #Temp_Str, N := 4, OUT => #BackData);
       #CheckSum := MID(IN := #返回数据, L := 4, P := 10);
       #求和 := 0;//..........................................................
       Strg_TO_Chars(Strg := #返回数据,
                     pChars := 0,
                     Cnt => #j,
                     Chars := #Temp_Chars);
       FOR #i := 1 TO 8 BY 1 DO
           #求和 := #求和 + #Temp_Chars[#i];
       END_FOR;
       #Temp_Word := DWORD_TO_WORD(#求和 MOD 65536);
       #Temp_Word := NOT #Temp_Word;
       #Temp_Word := #Temp_Word + 1; //Checksum
       #j := HTA(IN := #Temp_Word, N := 4, OUT => #Temp_Str);//Checksum明码.....
       IF #Temp_Str = #CheckSum THEN
           #喷码机数据返回 := 1;
       ELSE
           #喷码机数据返回 := 0;
       END_IF;
       #已满1000条 := 0;
       #不在喷印状态 := 0;
       #上一条信息没有喷完 := 0;
       IF #OrderID = 16#01 THEN
           IF #RTN = 16#00 THEN
               #数据条数 := #BackData;
           END_IF;
           IF #RTN = 16#02 THEN
               #已满1000条 := 1;
           END_IF;
           IF #RTN = 16#EF THEN
               #不在喷印状态 := 1;
           END_IF;
       END_IF;
       IF #OrderID = 16#02 THEN
           IF #RTN = 16#00 THEN
               #数据条数 := #BackData;
           END_IF;
           IF #RTN = 16#06 THEN
               #上一条信息没有喷完 := 1;
           END_IF;
           IF #RTN = 16#EF THEN
               #不在喷印状态 := 1;
           END_IF;
       END_IF;
       IF #OrderID = 16#03 THEN
           IF #RTN = 16#00 THEN
               #数据条数 := 0;
           END_IF;
           IF #RTN = 16#04 THEN
               #数据条数 := 0;
           END_IF;
       END_IF;
       IF #OrderID = 16#FE THEN
           IF #RTN = 16#00 THEN
               #数据条数 := #BackData;
           END_IF;
       END_IF;
   ELSE
       #喷码机数据返回 := 0;
   END_IF;
END_FUNCTION

// ===== library: MasterCopy "打包_01_Byte" =====

// folder: FC/位处理

FUNCTION "打包_01_Byte" : Byte   // FC10, SCL
{ S7_Optimized_Access := 'TRUE' }
VERSION : 0.1
   VAR_INPUT
      IN : Array[0..7] of Bool;
   END_VAR
   VAR_TEMP
      TempByte : Byte;
      i : Int;
   END_VAR
BEGIN
   #TempByte := BOOL_TO_BYTE(#IN[7]);
   FOR #i := 6 TO 0 BY -1 DO
       #TempByte := SHL(IN := #TempByte, N := 1);
       #TempByte := #TempByte + BOOL_TO_BYTE(#IN[#i]);
   END_FOR;
   #打包_01_Byte := #TempByte;
END_FUNCTION

// ===== library: MasterCopy "打包_02_Word" =====

// folder: FC/位处理

FUNCTION "打包_02_Word" : Word   // FC11, SCL
{ S7_Optimized_Access := 'TRUE' }
VERSION : 0.1
   VAR_INPUT
      IN : Array[0..15] of Bool;
   END_VAR
   VAR_TEMP
      TempWord : Word;
      i : Int;
   END_VAR
BEGIN
   #TempWord := BOOL_TO_WORD(#IN[15]);
   FOR #i := 14 TO 0 BY -1 DO
       #TempWord := SHL(IN := #TempWord, N := 1);
       #TempWord := #TempWord + BOOL_TO_WORD(#IN[#i]);
   END_FOR;
   #打包_02_Word := #TempWord;
END_FUNCTION

// ===== library: MasterCopy "解包_01_Byte" =====

// folder: FC/位处理

FUNCTION "解包_01_Byte" : Void   // FC12, SCL
{ S7_Optimized_Access := 'TRUE' }
VERSION : 0.1
   VAR_INPUT
      IN : Byte;
   END_VAR
   VAR_OUTPUT
      Out : Array[0..7] of Bool;
   END_VAR
   VAR_TEMP
      TempByte : Byte;
      i : Int;
   END_VAR
BEGIN
   #TempByte := #IN;
   #Out[0] := BYTE_TO_BOOL(#TempByte AND 1);
   FOR #i := 1 TO 7 BY 1 DO
       #TempByte := SHR(IN := #TempByte, N := 1);
       #Out[#i] := BYTE_TO_BOOL(#TempByte AND 1);
   END_FOR;
END_FUNCTION

// ===== library: MasterCopy "解包_02_Word" =====

// folder: FC/位处理

FUNCTION "解包_02_Word" : Void   // FC13, SCL
{ S7_Optimized_Access := 'TRUE' }
VERSION : 0.1
   VAR_INPUT
      IN : Word;
   END_VAR
   VAR_OUTPUT
      Out : Array[0..15] of Bool;
   END_VAR
   VAR_TEMP
      TempWord : Word;
      i : Int;
   END_VAR
BEGIN
   #TempWord := #IN;
   #Out[0] := WORD_TO_BOOL(#TempWord AND 1);
   FOR #i := 1 TO 15 BY 1 DO
       #TempWord := SHR(IN := #TempWord, N := 1);
       #Out[#i] := WORD_TO_BOOL(#TempWord AND 1);
   END_FOR;
END_FUNCTION

// ===== library: MasterCopy "MB_LSB_2W_R" =====

// folder: FC/小端数据组合

FUNCTION "MB_LSB_2W_R" : Void   // FC14, SCL
{ S7_Optimized_Access := 'TRUE' }
VERSION : 0.1
   VAR_INPUT
      "WORD" : Array[0..1] of Word;
   END_VAR
   VAR_OUTPUT
      Out : Real;
   END_VAR
   VAR_TEMP
      TempDword : DWord;
   END_VAR
BEGIN
   #TempDword := #WORD[1];
   #TempDword := SHL(IN := #TempDword, N := 16);
   #TempDword := #TempDword + #WORD[0];
   #Out := DWORD_TO_REAL(#TempDword);
END_FUNCTION

// ===== library: MasterCopy "MB_LSB_4B_R" =====

// folder: FC/小端数据组合

FUNCTION "MB_LSB_4B_R" : Void   // FC15, SCL
{ S7_Optimized_Access := 'TRUE' }
VERSION : 0.1
   VAR_INPUT
      "BYTE" : Array[0..3] of Byte;
   END_VAR
   VAR_OUTPUT
      Out : Real;
   END_VAR
   VAR_TEMP
      TempDword : DWord;
   END_VAR
BEGIN
   #TempDword := #BYTE[2];
   #TempDword := SHL(IN := #TempDword, N := 8);
   #TempDword := #TempDword + #BYTE[3];
   #TempDword := SHL(IN := #TempDword, N := 8);
   #TempDword := #TempDword + #BYTE[0];
   #TempDword := SHL(IN := #TempDword, N := 8);
   #TempDword := #TempDword + #BYTE[1];
   #Out := DWORD_TO_REAL(#TempDword);
END_FUNCTION